C07294=1020.176,319.167,359.790,170.598,49.800,159.708
C07295=1020.170,318.918,359.824,170.593,49.803,159.708
C07296=1020.163,318.671,359.858,170.586,49.806,159.708
C07297=1020.156,318.424,359.891,170.580,49.809,159.707
C07298=1020.149,318.176,359.925,170.574,49.812,159.707
C07299=1020.143,317.928,359.959,170.568,49.814,159.707
C07300=1020.136,317.681,359.993,170.563,49.818,159.706
C07301=1020.129,317.433,360.027,170.556,49.821,159.706
C07302=1020.122,317.186,360.060,170.551,49.823,159.706
C07303=1020.116,316.938,360.094,170.545,49.826,159.705
C07304=1020.109,316.690,360.128,170.538,49.829,159.705
C07305=1020.102,316.443,360.161,170.533,49.832,159.705
C07306=1020.095,316.195,360.195,170.527,49.835,159.705
C07307=1020.089,315.947,360.229,170.521,49.838,159.704
C07308=1020.083,315.700,360.262,170.515,49.840,159.704
C07309=1020.075,315.452,360.296,170.510,49.844,159.704
C07310=1020.069,315.205,360.329,170.503,49.847,159.704
C07311=1020.063,314.957,360.363,170.497,49.849,159.703
C07312=1020.056,314.710,360.396,170.492,49.853,159.703
C07313=1020.049,314.462,360.430,170.485,49.855,159.703
C07314=1020.042,314.214,360.463,170.480,49.858,159.702
C07315=1020.036,313.966,360.497,170.474,49.861,159.702
C07316=1020.030,313.719,360.530,170.468,49.864,159.702
C07317=1020.023,313.471,360.564,170.462,49.867,159.702
C07318=1020.016,313.224,360.597,170.457,49.870,159.702
C07319=1020.010,312.975,360.631,170.451,49.873,159.701
C07320=1020.003,312.729,360.665,170.445,49.877,159.701
C07321=1019.997,312.481,360.697,170.439,49.879,159.701
C07322=1019.990,312.233,360.731,170.434,49.883,159.701
C07323=1019.983,311.986,360.764,170.427,49.886,159.700
C07324=1019.978,311.738,360.798,170.422,49.889,159.700
C07325=1019.971,311.490,360.831,170.416,49.891,159.700
C07326=1019.964,311.243,360.865,170.411,49.895,159.700
C07327=1019.957,310.995,360.898,170.404,49.898,159.699
C07328=1019.952,310.747,360.931,170.399,49.901,159.699
C07329=1019.945,310.500,360.964,170.393,49.904,159.699
C07330=1019.938,310.252,360.998,170.388,49.907,159.699
C07331=1019.932,310.004,361.030,170.382,49.910,159.699
C07332=1019.925,309.757,361.064,170.376,49.913,159.698
C07333=1019.918,309.509,361.097,170.371,49.917,159.698
C07334=1019.911,309.262,361.129,170.365,49.920,159.698
C07335=1019.905,309.014,361.162,170.359,49.923,159.698
C07336=1019.897,308.766,361.194,170.353,49.927,159.698
C07337=1019.891,308.523,361.226,170.347,49.930,159.698
C07338=1019.885,308.281,361.258,170.342,49.933,159.697
C07339=1019.878,308.039,361.290,170.337,49.936,159.697
C07340=1019.871,307.796,361.322,170.332,49.940,159.697
C07341=1019.864,307.553,361.353,170.325,49.943,159.697
C07342=1019.858,307.311,361.385,170.320,49.947,159.697
C07343=1019.852,307.069,361.418,170.315,49.950,159.697
C07344=1019.845,306.827,361.449,170.309,49.953,159.697
C07345=1019.839,306.579,361.481,170.303,49.957,159.697
C07346=1019.831,306.331,361.514,170.298,49.960,159.696
C07347=1019.825,306.083,361.547,170.293,49.963,159.696
C07348=1019.819,305.836,361.579,170.286,49.967,159.696
C07349=1019.812,305.588,361.611,170.281,49.970,159.696
C07350=1019.806,305.340,361.643,170.276,49.974,159.696
C07351=1019.798,305.092,361.676,170.269,49.977,159.696
C07352=1019.792,304.845,361.709,170.264,49.981,159.696
C07353=1019.785,304.597,361.741,170.259,49.984,159.696
C07354=1019.779,304.349,361.773,170.253,49.987,159.695
C07355=1019.772,304.102,361.806,170.247,49.991,159.695
C07356=1019.765,303.854,361.838,170.242,49.995,159.695
C07357=1019.759,303.605,361.870,170.236,49.998,159.695
C07358=1019.752,303.358,361.903,170.231,50.002,159.695
C07359=1019.745,303.110,361.935,170.226,50.005,159.695
C07360=1019.739,302.862,361.967,170.219,50.009,159.695
C07361=1019.732,302.615,361.999,170.214,50.013,159.695
C07362=1019.726,302.367,362.031,170.209,50.016,159.695
C07363=1019.719,302.119,362.063,170.204,50.019,159.695
C07364=1019.713,301.872,362.096,170.198,50.023,159.694
C07365=1019.707,301.624,362.128,170.192,50.026,159.694
C07366=1019.699,301.376,362.161,170.187,50.030,159.694
C07367=1019.693,301.127,362.193,170.181,50.034,159.694
C07368=1019.686,300.880,362.225,170.176,50.037,159.694
C07369=1019.680,300.632,362.257,170.171,50.041,159.694
C07370=1019.674,300.384,362.288,170.165,50.045,159.694
C07371=1019.667,300.136,362.321,170.159,50.048,159.694
C07372=1019.661,299.888,362.353,170.154,50.052,159.694
C07373=1019.654,299.641,362.385,170.149,50.055,159.694
C07374=1019.648,299.393,362.417,170.143,50.059,159.694
C07375=1019.641,299.145,362.449,170.138,50.063,159.694
C07376=1019.635,298.897,362.481,170.133,50.066,159.694
C07377=1019.629,298.650,362.513,170.128,50.070,159.694
C07378=1019.623,298.402,362.545,170.121,50.074,159.694
C07379=1019.617,298.154,362.577,170.116,50.077,159.693
C07380=1019.610,297.906,362.609,170.111,50.081,159.694
C07381=1019.604,297.658,362.641,170.106,50.084,159.693
C07382=1019.597,297.411,362.673,170.100,50.089,159.693
C07383=1019.591,297.163,362.705,170.095,50.092,159.693
C07384=1019.585,296.915,362.736,170.090,50.096,159.693
C07385=1019.579,296.667,362.768,170.084,50.100,159.693
C07386=1019.572,296.419,362.801,170.079,50.104,159.693
C07387=1019.566,296.172,362.832,170.073,50.107,159.693
C07388=1019.560,295.924,362.864,170.069,50.111,159.693
C07389=1019.553,295.676,362.896,170.063,50.115,159.693
C07390=1019.547,295.427,362.928,170.057,50.118,159.693
C07391=1019.541,295.179,362.959,170.052,50.122,159.693
C07392=1019.535,294.933,362.991,170.047,50.126,159.693
C07393=1019.529,294.684,363.024,170.042,50.130,159.693
C07394=1019.522,294.436,363.055,170.036,50.134,159.693
C07395=1019.516,294.188,363.087,170.031,50.137,159.693
C07396=1019.510,293.940,363.118,170.026,50.141,159.693
C07397=1019.504,293.707,363.147,170.021,50.145,159.693
C07398=1019.499,293.473,363.178,170.016,50.149,159.693
C07399=1019.492,293.240,363.208,170.011,50.152,159.693
C07400=1019.486,293.006,363.238,170.006,50.156,159.693
C07401=1019.481,292.772,363.267,170.001,50.160,159.693
C07402=1019.475,292.539,363.297,169.996,50.163,159.693
C07403=1019.469,292.305,363.326,169.992,50.167,159.693
C07404=1019.462,292.072,363.356,169.987,50.171,159.693
C07405=1019.457,291.823,363.387,169.981,50.175,159.693
C07406=1019.450,291.575,363.418,169.976,50.179,159.694
C07407=1019.443,291.328,363.450,169.971,50.183,159.694
C07408=1019.437,291.080,363.481,169.965,50.187,159.694
C07409=1019.431,290.832,363.512,169.960,50.191,159.694
C07410=1019.424,290.584,363.543,169.955,50.195,159.694
C07411=1019.419,290.336,363.574,169.951,50.199,159.694
C07412=1019.412,290.088,363.605,169.945,50.204,159.694
C07413=1019.405,289.840,363.637,169.940,50.208,159.694
C07414=1019.400,289.592,363.667,169.935,50.212,159.694
C07415=1019.393,289.344,363.699,169.929,50.216,159.694
C07416=1019.386,289.096,363.729,169.924,50.220,159.694
C07417=1019.380,288.849,363.760,169.919,50.224,159.694
C07418=1019.374,288.601,363.792,169.913,50.228,159.694
C07419=1019.367,288.352,363.823,169.908,50.232,159.694
C07420=1019.361,288.105,363.854,169.903,50.236,159.694
C07421=1019.355,287.856,363.884,169.899,50.240,159.694
C07422=1019.348,287.608,363.916,169.893,50.245,159.694
C07423=1019.342,287.361,363.946,169.888,50.249,159.695
C07424=1019.336,287.112,363.977,169.883,50.253,159.695
C07425=1019.329,286.865,364.008,169.877,50.258,159.695
C07426=1019.323,286.616,364.039,169.872,50.262,159.695
C07427=1019.316,286.369,364.070,169.868,50.265,159.695
C07428=1019.311,286.121,364.100,169.863,50.270,159.695
C07429=1019.304,285.872,364.131,169.857,50.274,159.695
C07430=1019.298,285.625,364.162,169.852,50.278,159.695
C07431=1019.292,285.376,364.193,169.847,50.282,159.695
C07432=1019.286,285.129,364.223,169.842,50.287,159.696
C07433=1019.279,284.881,364.255,169.837,50.291,159.696
C07434=1019.273,284.633,364.285,169.832,50.295,159.696
C07435=1019.267,284.384,364.316,169.827,50.300,159.696
C07436=1019.261,284.137,364.346,169.822,50.304,159.696
C07437=1019.255,283.888,364.377,169.817,50.309,159.696
C07438=1019.248,283.641,364.407,169.811,50.313,159.696
C07439=1019.242,283.392,364.437,169.807,50.318,159.697
C07440=1019.235,283.145,364.468,169.802,50.322,159.697
C07441=1019.229,282.896,364.499,169.796,50.327,159.697
C07442=1019.222,282.649,364.529,169.791,50.331,159.697
C07443=1019.216,282.400,364.560,169.787,50.336,159.697
C07444=1019.210,282.152,364.590,169.782,50.340,159.697
C07445=1019.204,281.904,364.621,169.776,50.345,159.698
C07446=1019.197,281.656,364.650,169.772,50.349,159.698
C07447=1019.191,281.409,364.681,169.767,50.353,159.698
C07448=1019.185,281.160,364.711,169.761,50.358,159.698
C07449=1019.179,280.912,364.742,169.757,50.362,159.698
C07450=1019.173,280.664,364.772,169.752,50.366,159.698
C07451=1019.166,280.416,364.802,169.746,50.371,159.698
C07452=1019.160,280.168,364.833,169.742,50.376,159.699
C07453=1019.154,279.920,364.863,169.737,50.380,159.699
C07454=1019.148,279.671,364.893,169.731,50.385,159.699
C07455=1019.141,279.423,364.923,169.726,50.389,159.699
C07456=1019.136,279.175,364.953,169.722,50.394,159.699
C07457=1019.130,278.948,364.981,169.717,50.398,159.699
C07458=1019.124,278.721,365.009,169.713,50.402,159.700
C07459=1019.119,278.493,365.037,169.708,50.406,159.700
C07460=1019.113,278.265,365.064,169.704,50.411,159.700
C07461=1019.108,278.038,365.092,169.699,50.415,159.700
C07462=1019.102,277.810,365.120,169.694,50.419,159.700
C07463=1019.096,277.583,365.148,169.690,50.423,159.701
C07464=1019.090,277.355,365.175,169.685,50.427,159.701
C07465=1019.084,277.107,365.205,169.681,50.432,159.701
C07466=1019.079,276.859,365.235,169.676,50.437,159.701
C07467=1019.073,276.611,365.266,169.672,50.441,159.702
C07468=1019.066,276.363,365.295,169.666,50.446,159.702
C07469=1019.060,276.115,365.326,169.661,50.450,159.702
C07470=1019.054,275.867,365.355,169.657,50.455,159.702
C07471=1019.047,275.618,365.385,169.651,50.460,159.702
C07472=1019.041,275.371,365.415,169.647,50.465,159.703
C07473=1019.035,275.122,365.445,169.641,50.470,159.703
C07474=1019.029,274.875,365.475,169.637,50.475,159.703
C07475=1019.023,274.626,365.505,169.632,50.479,159.703
C07476=1019.016,274.378,365.534,169.627,50.484,159.704
C07477=1019.011,274.130,365.564,169.622,50.489,159.704
C07478=1019.004,273.882,365.594,169.618,50.494,159.704
C07479=1018.999,273.634,365.623,169.612,50.499,159.704
C07480=1018.991,273.385,365.653,169.608,50.503,159.705
C07481=1018.986,273.137,365.683,169.603,50.508,159.705
C07482=1018.979,272.889,365.713,169.598,50.513,159.705
C07483=1018.974,272.641,365.742,169.593,50.518,159.705
C07484=1018.968,272.393,365.771,169.589,50.522,159.706
C07485=1018.962,272.145,365.802,169.583,50.527,159.706
C07486=1018.955,271.896,365.831,169.579,50.532,159.706
C07487=1018.949,271.648,365.860,169.575,50.537,159.707
C07488=1018.943,271.400,365.891,169.569,50.542,159.707
C07489=1018.937,271.152,365.920,169.565,50.547,159.707
C07490=1018.931,270.904,365.949,169.560,50.552,159.707
C07491=1018.925,270.656,365.979,169.555,50.557,159.707
C07492=1018.918,270.408,366.008,169.550,50.562,159.708
C07493=1018.913,270.160,366.038,169.545,50.567,159.708
C07494=1018.906,269.911,366.067,169.540,50.572,159.708
C07495=1018.900,269.662,366.097,169.536,50.577,159.709
C07496=1018.894,269.415,366.127,169.530,50.582,159.709
C07497=1018.888,269.167,366.156,169.526,50.587,159.709
C07498=1018.882,268.918,366.185,169.522,50.592,159.710
C07499=1018.876,268.670,366.214,169.516,50.597,159.710
C07500=1018.870,268.422,366.243,169.512,50.602,159.710
C07501=1018.863,268.174,366.272,169.507,50.607,159.710
C07502=1018.858,267.925,366.302,169.502,50.612,159.711
C07503=1018.852,267.677,366.331,169.498,50.617,159.711
C07504=1018.845,267.429,366.360,169.493,50.622,159.711
C07505=1018.839,267.181,366.389,169.488,50.627,159.712
C07506=1018.834,266.933,366.419,169.484,50.632,159.712
C07507=1018.827,266.684,366.448,169.479,50.637,159.712
C07508=1018.821,266.436,366.477,169.474,50.643,159.713
C07509=1018.815,266.188,366.506,169.469,50.648,159.713
C07510=1018.809,265.940,366.535,169.465,50.653,159.714
C07511=1018.803,265.692,366.565,169.460,50.658,159.714
C07512=1018.797,265.443,366.594,169.455,50.664,159.714
C07513=1018.791,265.195,366.623,169.451,50.668,159.714
C07514=1018.784,264.947,366.652,169.446,50.674,159.715
C07515=1018.778,264.699,366.681,169.441,50.679,159.715
C07516=1018.772,264.451,366.710,169.437,50.684,159.716
C07517=1018.767,264.226,366.736,169.433,50.689,159.716
C07518=1018.762,264.000,366.762,169.428,50.693,159.716
C07519=1018.755,263.775,366.788,169.424,50.698,159.716
C07520=1018.750,263.550,366.815,169.419,50.703,159.717
C07521=1018.745,263.324,366.841,169.415,50.708,159.717
C07522=1018.739,263.099,366.866,169.412,50.713,159.718
C07523=1018.734,262.875,366.893,169.407,50.717,159.718
C07524=1018.728,262.649,366.919,169.403,50.722,159.718
C07525=1018.722,262.400,366.948,169.398,50.728,159.718
C07526=1018.717,262.153,366.977,169.393,50.733,159.719
C07527=1018.710,261.904,367.006,169.389,50.738,159.719
C07528=1018.704,261.656,367.034,169.384,50.744,159.720
C07529=1018.698,261.408,367.063,169.380,50.749,159.720
C07530=1018.692,261.159,367.093,169.375,50.755,159.720
C07531=1018.686,260.911,367.121,169.370,50.759,159.721
C07532=1018.680,260.662,367.150,169.366,50.765,159.721
C07533=1018.674,260.415,367.179,169.361,50.771,159.722
C07534=1018.668,260.166,367.207,169.357,50.776,159.722
C07535=1018.662,259.918,367.236,169.352,50.781,159.722
C07536=1018.656,259.669,367.264,169.347,50.786,159.723
C07537=1018.649,259.422,367.293,169.342,50.792,159.723
C07538=1018.643,259.173,367.321,169.338,50.798,159.724
C07539=1018.638,258.925,367.349,169.333,50.803,159.724
C07540=1018.631,258.677,367.377,169.329,50.809,159.724
C07541=1018.625,258.428,367.406,169.324,50.814,159.725
C07542=1018.619,258.179,367.434,169.320,50.820,159.725
C07543=1018.612,257.932,367.463,169.315,50.826,159.726
C07544=1018.606,257.683,367.491,169.311,50.832,159.726
C07545=1018.601,257.435,367.519,169.306,50.837,159.727
C07546=1018.594,257.187,367.547,169.301,50.843,159.727
C07547=1018.588,256.938,367.576,169.297,50.848,159.728
C07548=1018.582,256.690,367.604,169.292,50.854,159.728
C07549=1018.575,256.441,367.632,169.288,50.860,159.729
C07550=1018.570,256.193,367.660,169.283,50.865,159.729
C07551=1018.563,255.945,367.689,169.279,50.871,159.729
C07552=1018.557,255.696,367.716,169.273,50.877,159.730
C07553=1018.551,255.448,367.745,169.269,50.882,159.730
C07554=1018.545,255.200,367.773,169.265,50.888,159.731
C07555=1018.539,254.951,367.800,169.261,50.894,159.731
C07556=1018.533,254.703,367.829,169.256,50.900,159.732
C07557=1018.527,254.455,367.857,169.252,50.905,159.732
C07558=1018.521,254.207,367.885,169.246,50.911,159.733
C07559=1018.515,253.958,367.913,169.243,50.917,159.733
C07560=1018.508,253.709,367.941,169.238,50.923,159.734
C07561=1018.503,253.461,367.969,169.234,50.928,159.734
C07562=1018.497,253.213,367.997,169.229,50.934,159.734
C07563=1018.490,252.964,368.025,169.224,50.940,159.735
C07564=1018.485,252.716,368.053,169.220,50.946,159.736
C07565=1018.479,252.467,368.081,169.215,50.951,159.736
C07566=1018.472,252.220,368.110,169.211,50.957,159.736
C07567=1018.466,251.972,368.138,169.206,50.963,159.737
C07568=1018.460,251.723,368.166,169.202,50.969,159.737
C07569=1018.454,251.475,368.194,169.197,50.974,159.738
C07570=1018.448,251.226,368.222,169.193,50.980,159.738
C07571=1018.442,250.977,368.250,169.188,50.986,159.739
C07572=1018.436,250.730,368.278,169.184,50.992,159.739
C07573=1018.431,250.480,368.305,169.179,50.998,159.740
C07574=1018.425,250.233,368.333,169.175,51.003,159.740
C07575=1018.419,249.984,368.361,169.171,51.010,159.741
C07576=1018.413,249.735,368.389,169.167,51.015,159.741
C07577=1018.407,249.510,368.414,169.163,51.021,159.742
C07578=1018.402,249.284,368.440,169.158,51.026,159.742
C07579=1018.396,249.057,368.465,169.154,51.032,159.743
C07580=1018.392,248.831,368.491,169.150,51.037,159.743
C07581=1018.386,248.605,368.516,169.146,51.042,159.744
C07582=1018.381,248.379,368.541,169.142,51.048,159.744
C07583=1018.375,248.154,368.566,169.138,51.053,159.745
C07584=1018.370,247.927,368.592,169.134,51.059,159.745
C07585=1018.364,247.679,368.620,169.129,51.065,159.746
C07586=1018.358,247.430,368.647,169.125,51.071,159.746
C07587=1018.353,247.182,368.675,169.120,51.076,159.747
C07588=1018.346,246.934,368.703,169.117,51.083,159.747
C07589=1018.341,246.685,368.731,169.112,51.088,159.748
C07590=1018.334,246.437,368.759,169.108,51.094,159.748
C07591=1018.329,246.188,368.786,169.103,51.100,159.749
C07592=1018.323,245.940,368.814,169.098,51.107,159.749
C07593=1018.317,245.692,368.842,169.094,51.112,159.750
C07594=1018.311,245.443,368.869,169.090,51.119,159.750
C07595=1018.306,245.194,368.897,169.085,51.124,159.751
C07596=1018.300,244.947,368.925,169.081,51.130,159.751
C07597=1018.294,244.698,368.953,169.077,51.137,159.752
C07598=1018.288,244.450,368.979,169.072,51.142,159.753
C07599=1018.282,244.201,369.008,169.068,51.148,159.753
C07600=1018.277,243.953,369.036,169.064,51.155,159.754
C07601=1018.271,243.704,369.062,169.060,51.160,159.754
C07602=1018.265,243.456,369.091,169.055,51.167,159.755
C07603=1018.259,243.208,369.118,169.050,51.173,159.755
C07604=1018.254,242.959,369.146,169.046,51.179,159.756
C07605=1018.247,242.711,369.173,169.042,51.185,159.756
C07606=1018.242,242.462,369.200,169.038,51.191,159.757
C07607=1018.236,242.214,369.228,169.034,51.198,159.758
C07608=1018.230,241.965,369.255,169.029,51.204,159.758
C07609=1018.222,241.657,369.289,169.024,51.212,159.759
C07610=1018.216,241.348,369.323,169.018,51.219,159.760
C07611=1018.208,241.040,369.357,169.014,51.227,159.761
C07612=1018.201,240.731,369.390,169.007,51.235,159.761
C07613=1018.195,240.483,369.418,169.004,51.241,159.762
C07614=1018.189,240.233,369.445,168.999,51.248,159.762
C07615=1018.183,239.985,369.472,168.994,51.254,159.763
C07616=1018.177,239.737,369.499,168.991,51.261,159.764
C07617=1018.172,239.489,369.526,168.986,51.267,159.764
C07618=1018.166,239.240,369.553,168.981,51.274,159.765
C07619=1018.160,238.992,369.581,168.978,51.280,159.766
C07620=1018.154,238.743,369.607,168.973,51.286,159.766
C07621=1018.148,238.494,369.634,168.969,51.293,159.767
C07622=1018.143,238.246,369.662,168.965,51.299,159.767
C07623=1018.137,237.998,369.689,168.960,51.305,159.768
C07624=1018.130,237.749,369.716,168.956,51.312,159.769
C07625=1018.124,237.501,369.743,168.951,51.318,159.769
C07626=1018.119,237.252,369.769,168.947,51.324,159.770
C07627=1018.113,237.004,369.796,168.943,51.332,159.771
C07628=1018.107,236.755,369.823,168.939,51.338,159.771
C07629=1018.101,236.506,369.850,168.934,51.345,159.772
C07630=1018.095,236.258,369.876,168.930,51.351,159.772
C07631=1018.089,236.010,369.903,168.926,51.357,159.773
C07632=1018.083,235.761,369.931,168.921,51.364,159.774
C07633=1018.077,235.513,369.957,168.918,51.371,159.775
C07634=1018.071,235.265,369.984,168.913,51.377,159.775
C07635=1018.065,235.016,370.011,168.909,51.384,159.776
C07636=1018.059,234.767,370.038,168.904,51.391,159.776
C07637=1018.049,234.368,370.080,168.897,51.401,159.777
C07638=1018.040,233.970,370.124,168.891,51.412,159.779
C07639=1018.031,233.571,370.166,168.884,51.422,159.780
C07640=1018.022,233.173,370.208,168.877,51.433,159.781
C07641=1018.015,232.924,370.235,168.873,51.440,159.781
C07642=1018.010,232.676,370.261,168.868,51.447,159.782
C07643=1018.004,232.428,370.288,168.865,51.453,159.783
C07644=1017.998,232.179,370.315,168.861,51.460,159.784
C07645=1017.992,231.931,370.341,168.856,51.466,159.784
C07646=1017.986,231.682,370.368,168.852,51.474,159.785
C07647=1017.981,231.434,370.395,168.847,51.480,159.785
C07648=1017.975,231.184,370.421,168.844,51.487,159.786
C07649=1017.969,230.936,370.448,168.839,51.494,159.787
C07650=1017.963,230.688,370.474,168.835,51.500,159.788
C07651=1017.957,230.439,370.501,168.831,51.507,159.788
C07652=1017.952,230.191,370.528,168.826,51.514,159.789
C07653=1017.946,229.942,370.553,168.823,51.521,159.790
C07654=1017.940,229.694,370.580,168.818,51.527,159.790
C07655=1017.935,229.445,370.607,168.814,51.534,159.791
C07656=1017.929,229.197,370.633,168.810,51.542,159.792
C07657=1017.923,228.948,370.659,168.805,51.548,159.792
C07658=1017.917,228.700,370.685,168.802,51.555,159.793
C07659=1017.911,228.452,370.712,168.797,51.562,159.794
C07660=1017.906,228.203,370.738,168.793,51.569,159.795
C07661=1017.899,227.953,370.765,168.789,51.576,159.796
C07662=1017.893,227.705,370.792,168.784,51.582,159.796
C07663=1017.887,227.456,370.817,168.780,51.590,159.797
C07664=1017.881,227.208,370.844,168.776,51.597,159.798
C07665=1017.876,226.959,370.870,168.772,51.603,159.798
C07666=1017.870,226.711,370.896,168.768,51.610,159.799
C07667=1017.864,226.462,370.923,168.764,51.618,159.800
C07668=1017.858,226.214,370.948,168.760,51.625,159.801
C07669=1017.852,225.965,370.975,168.756,51.632,159.802
C07670=1017.846,225.717,371.000,168.751,51.639,159.802
C07671=1017.841,225.468,371.026,168.747,51.646,159.803
C07672=1017.835,225.219,371.053,168.743,51.653,159.804
C07673=1017.829,224.971,371.078,168.739,51.660,159.804
C07674=1017.823,224.722,371.105,168.734,51.667,159.805
C07675=1017.817,224.474,371.130,168.730,51.675,159.806
C07676=1017.811,224.225,371.156,168.726,51.682,159.807
C07677=1017.806,223.976,371.183,168.723,51.689,159.808
C07678=1017.799,223.728,371.208,168.719,51.696,159.809
C07679=1017.794,223.479,371.234,168.714,51.703,159.809
C07680=1017.788,223.231,371.260,168.710,51.710,159.810
C07681=1017.782,222.982,371.286,168.706,51.717,159.811
C07682=1017.776,222.734,371.311,168.702,51.724,159.811
C07683=1017.771,222.485,371.338,168.698,51.732,159.812
C07684=1017.765,222.236,371.363,168.693,51.739,159.813
C07685=1017.759,221.988,371.389,168.689,51.746,159.814
C07686=1017.753,221.739,371.415,168.685,51.753,159.815
C07687=1017.747,221.491,371.441,168.681,51.761,159.815
C07688=1017.741,221.242,371.467,168.677,51.768,159.816
C07689=1017.735,220.993,371.492,168.673,51.775,159.817
C07690=1017.729,220.745,371.519,168.669,51.783,159.818
C07691=1017.725,220.496,371.544,168.665,51.790,159.819
C07692=1017.718,220.248,371.570,168.661,51.798,159.820
C07693=1017.712,220.014,371.594,168.657,51.804,159.820
C07694=1017.707,219.781,371.618,168.653,51.811,159.821
C07695=1017.702,219.548,371.642,168.649,51.818,159.822
C07696=1017.697,219.313,371.667,168.645,51.824,159.822
C07697=1017.691,219.080,371.691,168.641,51.832,159.823
C07698=1017.686,218.847,371.715,168.638,51.839,159.824
C07699=1017.681,218.613,371.739,168.633,51.845,159.825
C07700=1017.675,218.379,371.764,168.630,51.852,159.826
C07701=1017.669,218.131,371.790,168.626,51.859,159.826
C07702=1017.664,217.883,371.815,168.622,51.867,159.827
C07703=1017.657,217.634,371.840,168.617,51.875,159.828
C07704=1017.651,217.385,371.865,168.613,51.882,159.829
C07705=1017.646,217.136,371.891,168.609,51.890,159.830
C07706=1017.640,216.888,371.916,168.605,51.897,159.831
C07707=1017.634,216.640,371.942,168.601,51.905,159.831
C07708=1017.628,216.391,371.967,168.597,51.913,159.832
C07709=1017.622,216.142,371.993,168.593,51.920,159.833
C07710=1017.616,215.893,372.018,168.589,51.927,159.834
C07711=1017.610,215.645,372.043,168.585,51.935,159.835
C07712=1017.605,215.396,372.068,168.581,51.942,159.836
C07713=1017.599,215.147,372.094,168.576,51.951,159.837
C07714=1017.593,214.898,372.119,168.572,51.958,159.838
C07715=1017.587,214.650,372.144,168.569,51.966,159.839
C07716=1017.582,214.401,372.170,168.565,51.973,159.839
C07717=1017.576,214.153,372.195,168.561,51.981,159.840
C07718=1017.569,213.904,372.221,168.557,51.989,159.841
C07719=1017.564,213.656,372.246,168.553,51.996,159.842
C07720=1017.559,213.407,372.271,168.549,52.004,159.843
C07721=1017.552,213.158,372.296,168.544,52.012,159.844
C07722=1017.546,212.909,372.321,168.540,52.019,159.845
C07723=1017.541,212.661,372.347,168.536,52.027,159.846
C07724=1017.535,212.412,372.372,168.532,52.035,159.846
C07725=1017.529,212.163,372.397,168.529,52.043,159.847
C07726=1017.524,211.915,372.422,168.524,52.050,159.848
C07727=1017.518,211.666,372.448,168.521,52.058,159.849
C07728=1017.512,211.417,372.473,168.516,52.066,159.850
C07729=1017.507,211.169,372.497,168.512,52.074,159.851
C07730=1017.500,210.920,372.523,168.508,52.082,159.852
C07731=1017.495,210.671,372.549,168.504,52.089,159.853
C07732=1017.489,210.423,372.574,168.500,52.097,159.854
C07733=1017.483,210.174,372.598,168.496,52.104,159.854
C07734=1017.477,209.925,372.624,168.493,52.112,159.855
C07735=1017.472,209.677,372.649,168.488,52.121,159.856
C07736=1017.466,209.428,372.674,168.484,52.128,159.857
C07737=1017.461,209.180,372.699,168.480,52.136,159.858
C07738=1017.455,208.930,372.723,168.477,52.144,159.859
C07739=1017.449,208.682,372.749,168.472,52.152,159.860
C07740=1017.443,208.434,372.774,168.468,52.160,159.861
C07741=1017.437,208.184,372.798,168.464,52.168,159.862
C07742=1017.431,207.936,372.824,168.460,52.176,159.863
C07743=1017.426,207.687,372.848,168.456,52.184,159.864
C07744=1017.420,207.438,372.873,168.452,52.192,159.865
C07745=1017.414,207.190,372.898,168.448,52.200,159.866
C07746=1017.408,206.941,372.923,168.445,52.208,159.867
C07747=1017.403,206.693,372.947,168.440,52.216,159.868
C07748=1017.397,206.444,372.972,168.436,52.224,159.868
C07749=1017.391,206.195,372.997,168.432,52.232,159.869
C07750=1017.385,205.947,373.022,168.429,52.240,159.870
C07751=1017.379,205.697,373.047,168.424,52.248,159.871
C07752=1017.374,205.449,373.071,168.420,52.256,159.872
C07753=1017.369,205.212,373.095,168.417,52.264,159.873
C07754=1017.362,204.975,373.118,168.413,52.271,159.874
C07755=1017.357,204.739,373.141,168.409,52.280,159.875
C07756=1017.352,204.503,373.164,168.405,52.288,159.876
C07757=1017.346,204.265,373.188,168.401,52.295,159.877
C07758=1017.340,204.029,373.211,168.398,52.303,159.878
C07759=1017.335,203.793,373.235,168.394,52.311,159.879
C07760=1017.330,203.556,373.258,168.390,52.319,159.880
C07761=1017.305,202.315,373.374,167.903,52.236,159.767
C07762=1017.300,202.066,373.396,167.898,52.246,159.768
C07763=1017.296,201.818,373.419,167.894,52.255,159.769
C07764=1017.291,201.570,373.442,167.889,52.264,159.770
C07765=1017.286,201.321,373.465,167.884,52.273,159.771
C07766=1017.281,201.072,373.487,167.880,52.282,159.772
C07767=1017.276,200.823,373.511,167.875,52.291,159.773
C07768=1017.272,200.573,373.533,167.870,52.301,159.774
C07769=1017.267,200.325,373.556,167.866,52.310,159.775
C07770=1017.262,200.077,373.579,167.861,52.319,159.776
C07771=1017.257,199.827,373.602,167.857,52.329,159.778
C07772=1017.253,199.578,373.625,167.852,52.338,159.779
C07773=1017.248,199.329,373.647,167.848,52.348,159.780
C07774=1017.243,199.080,373.671,167.843,52.357,159.781
C07775=1017.238,198.831,373.693,167.838,52.366,159.782
C07776=1017.233,198.583,373.715,167.834,52.376,159.783
C07777=1017.229,198.333,373.738,167.829,52.385,159.784
C07778=1017.223,198.085,373.761,167.825,52.395,159.785
C07779=1017.218,197.836,373.783,167.820,52.405,159.786
C07780=1017.214,197.587,373.805,167.816,52.414,159.787
C07781=1017.208,197.338,373.828,167.811,52.423,159.788
C07782=1017.203,197.089,373.850,167.806,52.433,159.789
C07783=1017.199,196.840,373.872,167.802,52.442,159.790
C07784=1017.194,196.591,373.895,167.797,52.452,159.791
C07785=1017.189,196.342,373.917,167.793,52.461,159.792
C07786=1017.184,196.093,373.939,167.789,52.471,159.794
C07787=1017.179,195.844,373.963,167.784,52.480,159.795
C07788=1017.174,195.595,373.985,167.780,52.490,159.796
C07789=1017.169,195.346,374.006,167.776,52.499,159.797
C07790=1017.165,195.097,374.029,167.770,52.509,159.798
C07791=1017.159,194.848,374.052,167.766,52.518,159.799
C07792=1017.155,194.600,374.074,167.762,52.528,159.800
C07793=1017.151,194.350,374.096,167.757,52.537,159.801
C07794=1017.145,194.101,374.118,167.753,52.547,159.802
C07795=1017.140,193.853,374.141,167.749,52.557,159.803
C07796=1017.135,193.604,374.163,167.744,52.566,159.804
C07797=1017.131,193.355,374.185,167.739,52.575,159.805
C07798=1017.126,193.105,374.207,167.736,52.585,159.807
C07799=1017.121,192.856,374.229,167.730,52.595,159.807
C07800=1017.117,192.607,374.252,167.726,52.604,159.809
C07801=1017.112,192.359,374.274,167.722,52.613,159.810
C07802=1017.106,192.110,374.297,167.718,52.623,159.811
C07803=1017.101,191.861,374.318,167.713,52.632,159.812
C07804=1017.097,191.612,374.341,167.709,52.642,159.813
C07805=1017.092,191.363,374.363,167.705,52.651,159.814
C07806=1017.088,191.114,374.385,167.701,52.661,159.815
C07807=1017.083,190.864,374.407,167.695,52.670,159.816
C07808=1017.078,190.615,374.429,167.692,52.680,159.817
C07809=1017.073,190.367,374.452,167.687,52.689,159.818
C07810=1017.069,190.118,374.474,167.683,52.698,159.819
C07811=1017.064,189.869,374.496,167.678,52.709,159.821
C07812=1017.059,189.620,374.518,167.674,52.718,159.822
C07813=1017.054,189.372,374.540,167.670,52.727,159.823
C07814=1017.050,189.122,374.563,167.666,52.737,159.824
C07815=1017.045,188.873,374.585,167.661,52.747,159.825
C07816=1017.040,188.624,374.607,167.657,52.756,159.826
C07817=1017.035,188.375,374.628,167.653,52.766,159.827
C07818=1017.031,188.126,374.651,167.649,52.775,159.828
C07819=1017.026,187.877,374.673,167.645,52.784,159.829
C07820=1017.022,187.629,374.695,167.640,52.794,159.830
C07821=1017.017,187.348,374.720,167.635,52.805,159.832
C07822=1017.011,187.068,374.745,167.631,52.816,159.833
C07823=1017.007,186.787,374.769,167.626,52.826,159.834
C07824=1017.001,186.507,374.794,167.622,52.837,159.836
C07825=1016.996,186.258,374.815,167.616,52.847,159.836
C07826=1016.992,186.009,374.837,167.612,52.856,159.838
C07827=1016.987,185.760,374.860,167.608,52.866,159.839
C07828=1016.983,185.511,374.881,167.604,52.875,159.840
C07829=1016.978,185.262,374.903,167.600,52.884,159.841
C07830=1016.974,185.013,374.926,167.596,52.894,159.842
C07831=1016.969,184.764,374.948,167.592,52.903,159.843
C07832=1016.964,184.516,374.970,167.588,52.913,159.844
C07833=1016.959,184.267,374.991,167.583,52.923,159.845
C07834=1016.955,184.017,375.013,167.579,52.932,159.846
C07835=1016.951,183.768,375.035,167.575,52.941,159.847
C07836=1016.946,183.519,375.057,167.571,52.951,159.849
C07837=1016.941,183.270,375.079,167.567,52.961,159.850
C07838=1016.937,183.021,375.101,167.563,52.970,159.851
C07839=1016.932,182.772,375.122,167.559,52.980,159.852
C07840=1016.928,182.523,375.144,167.555,52.989,159.853
C07841=1016.924,182.274,375.167,167.551,52.998,159.854
C07842=1016.919,182.025,375.189,167.547,53.008,159.856
C07843=1016.914,181.776,375.210,167.543,53.017,159.857
C07844=1016.909,181.527,375.232,167.538,53.028,159.858
C07845=1016.904,181.278,375.252,167.534,53.037,159.859
C07846=1016.899,181.029,375.274,167.530,53.047,159.860
C07847=1016.895,180.780,375.295,167.526,53.057,159.861
C07848=1016.889,180.530,375.316,167.522,53.067,159.862
C07849=1016.885,180.282,375.338,167.518,53.077,159.864
C07850=1016.880,180.032,375.359,167.514,53.086,159.865
C07851=1016.875,179.784,375.380,167.509,53.096,159.866
C07852=1016.870,179.534,375.401,167.505,53.106,159.867
C07853=1016.865,179.285,375.422,167.501,53.115,159.868
C07854=1016.860,179.036,375.444,167.498,53.125,159.869
C07855=1016.855,178.787,375.465,167.493,53.136,159.871
C07856=1016.850,178.538,375.485,167.489,53.145,159.872
C07857=1016.845,178.289,375.507,167.485,53.155,159.873
C07858=1016.841,178.039,375.528,167.481,53.165,159.874
C07859=1016.836,177.790,375.549,167.477,53.174,159.875
C07860=1016.831,177.542,375.571,167.473,53.185,159.876
C07861=1016.826,177.293,375.591,167.469,53.195,159.878
C07862=1016.822,177.044,375.612,167.465,53.204,159.879
C07863=1016.817,176.794,375.633,167.461,53.214,159.880
C07864=1016.812,176.546,375.654,167.457,53.224,159.881
C07865=1016.807,176.296,375.676,167.452,53.234,159.882
C07866=1016.803,176.047,375.697,167.449,53.244,159.883
C07867=1016.797,175.798,375.717,167.445,53.254,159.885
C07868=1016.792,175.549,375.739,167.441,53.263,159.886
C07869=1016.788,175.301,375.759,167.437,53.273,159.887
C07870=1016.783,175.051,375.780,167.434,53.283,159.888
C07871=1016.779,174.802,375.802,167.428,53.293,159.889
C07872=1016.773,174.553,375.822,167.425,53.303,159.891
C07873=1016.769,174.304,375.844,167.421,53.312,159.892
C07874=1016.763,174.055,375.865,167.417,53.322,159.893
C07875=1016.759,173.806,375.885,167.414,53.332,159.894
C07876=1016.755,173.556,375.907,167.409,53.341,159.895
C07877=1016.750,173.307,375.927,167.406,53.351,159.896
C07878=1016.745,173.058,375.948,167.401,53.362,159.898
C07879=1016.740,172.809,375.969,167.397,53.371,159.899
C07880=1016.736,172.561,375.990,167.393,53.381,159.900
C07881=1016.731,172.311,376.011,167.390,53.391,159.901
C07882=1016.726,172.062,376.032,167.386,53.400,159.902
C07883=1016.721,171.813,376.053,167.382,53.410,159.904
C07884=1016.718,171.564,376.074,167.378,53.420,159.905
C07885=1016.712,171.283,376.097,167.374,53.431,159.906
C07886=1016.707,171.003,376.121,167.370,53.442,159.907
C07887=1016.701,170.722,376.144,167.366,53.453,159.909
C07888=1016.695,170.441,376.168,167.360,53.465,159.910
C07889=1016.692,170.192,376.188,167.356,53.474,159.911
C07890=1016.687,169.943,376.210,167.353,53.484,159.912
C07891=1016.681,169.694,376.231,167.349,53.494,159.914
C07892=1016.678,169.445,376.252,167.345,53.503,159.915
C07893=1016.672,169.196,376.272,167.341,53.513,159.916
C07894=1016.668,168.947,376.293,167.338,53.524,159.917
C07895=1016.664,168.698,376.314,167.334,53.533,159.918
C07896=1016.659,168.449,376.335,167.330,53.543,159.920
C07897=1016.654,168.199,376.356,167.326,53.552,159.921
C07898=1016.649,167.951,376.376,167.323,53.562,159.922
C07899=1016.645,167.702,376.397,167.319,53.572,159.923
C07900=1016.641,167.452,376.417,167.315,53.582,159.924
C07901=1016.636,167.203,376.438,167.311,53.592,159.926
C07902=1016.631,166.954,376.459,167.307,53.601,159.927
C07903=1016.626,166.705,376.479,167.304,53.611,159.928
C07904=1016.622,166.456,376.500,167.300,53.621,159.929
C07905=1016.618,166.206,376.521,167.296,53.631,159.930
C07906=1016.613,165.957,376.542,167.293,53.641,159.932
C07907=1016.609,165.709,376.563,167.289,53.650,159.933
C07908=1016.603,165.459,376.583,167.285,53.660,159.934
C07909=1016.599,165.211,376.604,167.281,53.670,159.935
C07910=1016.594,164.962,376.625,167.278,53.680,159.936
C07911=1016.590,164.712,376.646,167.274,53.690,159.938
C07912=1016.586,164.463,376.666,167.270,53.699,159.939
C07913=1016.581,164.214,376.686,167.266,53.709,159.940
C07914=1016.577,163.965,376.707,167.262,53.719,159.941
C07915=1016.572,163.716,376.728,167.259,53.729,159.942
C07916=1016.567,163.466,376.749,167.255,53.739,159.944
C07917=1016.563,163.218,376.770,167.251,53.748,159.945
C07918=1016.558,162.968,376.789,167.249,53.758,159.946
C07919=1016.554,162.719,376.810,167.245,53.767,159.947
C07920=1016.549,162.470,376.831,167.241,53.778,159.948
C07921=1016.545,162.221,376.851,167.237,53.787,159.950
C07922=1016.541,161.972,376.873,167.234,53.797,159.951
C07923=1016.536,161.723,376.892,167.230,53.806,159.952
C07924=1016.532,161.473,376.913,167.226,53.817,159.953
C07925=1016.527,161.225,376.933,167.223,53.827,159.954
C07926=1016.523,160.976,376.955,167.219,53.836,159.956
C07927=1016.518,160.726,376.974,167.215,53.846,159.957
C07928=1016.514,160.477,376.995,167.212,53.855,159.958
C07929=1016.510,160.228,377.016,167.209,53.865,159.959
C07930=1016.505,159.979,377.037,167.205,53.875,159.960
C07931=1016.501,159.730,377.057,167.201,53.885,159.962
C07932=1016.496,159.481,377.077,167.197,53.894,159.963
C07933=1016.492,159.232,377.098,167.194,53.904,159.964
C07934=1016.487,158.982,377.118,167.190,53.914,159.965
C07935=1016.483,158.733,377.139,167.186,53.924,159.966
C07936=1016.478,158.484,377.160,167.184,53.933,159.968
C07937=1016.474,158.235,377.179,167.180,53.943,159.969
C07938=1016.469,157.986,377.200,167.177,53.953,159.970
C07939=1016.464,157.737,377.219,167.173,53.964,159.971
C07940=1016.459,157.488,377.240,167.169,53.973,159.973
C07941=1016.455,157.239,377.259,167.166,53.983,159.974
C07942=1016.450,156.989,377.279,167.162,53.993,159.975
C07943=1016.445,156.741,377.299,167.159,54.003,159.976
C07944=1016.441,156.490,377.320,167.155,54.014,159.978
C07945=1016.436,156.242,377.340,167.151,54.023,159.979
C07946=1016.432,155.993,377.359,167.148,54.033,159.980
C07947=1016.427,155.743,377.379,167.144,54.043,159.981
C07948=1016.422,155.495,377.399,167.141,54.053,159.983
C07949=1016.417,155.213,377.422,167.137,54.065,159.984
C07950=1016.412,154.932,377.444,167.133,54.076,159.986
C07951=1016.407,154.652,377.467,167.129,54.087,159.987
C07952=1016.402,154.371,377.489,167.125,54.098,159.988
C07953=1016.397,154.122,377.509,167.121,54.108,159.989
C07954=1016.392,153.873,377.529,167.118,54.118,159.991
C07955=1016.387,153.623,377.549,167.114,54.128,159.992
C07956=1016.383,153.375,377.569,167.110,54.138,159.993
C07957=1016.378,153.126,377.588,167.107,54.148,159.994
C07958=1016.374,152.876,377.608,167.103,54.158,159.996
C07959=1016.370,152.626,377.628,167.100,54.168,159.997
C07960=1016.364,152.378,377.648,167.096,54.178,159.998
C07961=1016.360,152.129,377.668,167.094,54.188,159.999
C07962=1016.355,151.880,377.687,167.090,54.198,160.001
C07963=1016.350,151.630,377.707,167.087,54.208,160.002
C07964=1016.346,151.381,377.726,167.083,54.218,160.003
C07965=1016.341,151.131,377.746,167.080,54.228,160.005
C07966=1016.336,150.883,377.766,167.076,54.238,160.006
C07967=1016.332,150.634,377.786,167.073,54.248,160.007
C07968=1016.327,150.384,377.806,167.069,54.258,160.008
C07969=1016.323,150.135,377.825,167.066,54.268,160.010
C07970=1016.318,149.886,377.845,167.062,54.278,160.011
C07971=1016.313,149.636,377.865,167.058,54.288,160.012
C07972=1016.309,149.387,377.884,167.055,54.298,160.013
C07973=1016.305,149.138,377.904,167.052,54.308,160.015
C07974=1016.299,148.889,377.924,167.048,54.318,160.016
C07975=1016.295,148.640,377.944,167.045,54.328,160.017
C07976=1016.291,148.391,377.963,167.042,54.338,160.019
C07977=1016.286,148.142,377.982,167.039,54.348,160.020
C07978=1016.281,147.892,378.002,167.035,54.358,160.021
C07979=1016.276,147.643,378.021,167.031,54.368,160.022
C07980=1016.272,147.394,378.041,167.028,54.378,160.024
C07981=1016.267,147.144,378.061,167.025,54.388,160.025
C07982=1016.263,146.895,378.080,167.021,54.399,160.026
C07983=1016.258,146.646,378.099,167.017,54.408,160.027
C07984=1016.254,146.397,378.119,167.014,54.418,160.029
C07985=1016.249,146.147,378.139,167.012,54.428,160.030
C07986=1016.244,145.899,378.158,167.008,54.438,160.031
C07987=1016.240,145.650,378.177,167.005,54.449,160.033
C07988=1016.235,145.401,378.197,167.001,54.458,160.034
C07989=1016.230,145.151,378.216,166.998,54.468,160.035
C07990=1016.226,144.901,378.235,166.994,54.479,160.036
C07991=1016.221,144.653,378.254,166.991,54.489,160.038
C07992=1016.217,144.403,378.274,166.988,54.499,160.039
C07993=1016.212,144.154,378.293,166.984,54.509,160.040
C07994=1016.207,143.905,378.312,166.981,54.519,160.041
C07995=1016.202,143.656,378.332,166.977,54.529,160.043
C07996=1016.198,143.406,378.350,166.975,54.539,160.044
C07997=1016.193,143.157,378.370,166.972,54.549,160.045
C07998=1016.188,142.908,378.389,166.968,54.560,160.047
C07999=1016.184,142.659,378.409,166.965,54.570,160.048
C08000=1016.179,142.409,378.427,166.962,54.580,160.049
C08001=1016.175,142.160,378.446,166.958,54.590,160.050
C08002=1016.170,141.911,378.466,166.954,54.600,160.052
C08003=1016.165,141.662,378.485,166.951,54.610,160.053
C08004=1016.161,141.413,378.504,166.948,54.620,160.054
C08005=1016.156,141.163,378.523,166.946,54.630,160.056
C08006=1016.151,140.914,378.542,166.942,54.640,160.057
C08007=1016.146,140.665,378.562,166.938,54.650,160.058
C08008=1016.142,140.415,378.581,166.935,54.660,160.060
C08009=1016.137,140.166,378.600,166.932,54.671,160.061
C08010=1016.133,139.917,378.619,166.928,54.681,160.062
C08011=1016.129,139.668,378.639,166.925,54.690,160.063
C08012=1016.124,139.419,378.657,166.922,54.700,160.065
C08013=1016.119,139.138,378.679,166.919,54.712,160.066
C08014=1016.114,138.857,378.701,166.915,54.723,160.068
C08015=1016.108,138.576,378.721,166.911,54.734,160.069
C08016=1016.103,138.295,378.743,166.907,54.746,160.071
C08017=1016.099,138.046,378.763,166.905,54.756,160.072
C08018=1016.094,137.797,378.781,166.902,54.766,160.073
C08019=1016.089,137.547,378.801,166.898,54.776,160.075
C08020=1016.084,137.298,378.819,166.895,54.787,160.076
C08021=1016.080,137.048,378.838,166.891,54.796,160.077
C08022=1016.075,136.800,378.857,166.888,54.807,160.078
C08023=1016.071,136.550,378.876,166.885,54.817,160.080
C08024=1016.066,136.301,378.895,166.882,54.827,160.081
C08025=1016.062,136.052,378.914,166.879,54.837,160.083
C08026=1016.057,135.803,378.932,166.876,54.847,160.084
C08027=1016.053,135.553,378.951,166.872,54.857,160.085
C08028=1016.047,135.305,378.970,166.869,54.867,160.086
C08029=1016.043,135.054,378.989,166.866,54.878,160.088
C08030=1016.038,134.805,379.008,166.862,54.888,160.089
C08031=1016.033,134.556,379.026,166.860,54.898,160.090
C08032=1016.029,134.306,379.045,166.857,54.908,160.092
C08033=1016.024,134.058,379.064,166.854,54.918,160.093
C08034=1016.020,133.808,379.083,166.850,54.928,160.094
C08035=1016.015,133.559,379.101,166.847,54.938,160.095
C08036=1016.010,133.310,379.120,166.843,54.949,160.097
C08037=1016.006,133.060,379.138,166.840,54.959,160.098
C08038=1016.001,132.812,379.157,166.838,54.969,160.100
C08039=1015.997,132.562,379.176,166.835,54.979,160.101
C08040=1015.992,132.313,379.195,166.831,54.989,160.102
C08041=1015.987,132.064,379.213,166.828,54.999,160.103
C08042=1015.983,131.814,379.232,166.825,55.010,160.105
C08043=1015.978,131.565,379.251,166.822,55.019,160.106
C08044=1015.973,131.316,379.269,166.819,55.030,160.108
C08045=1015.969,131.066,379.288,166.815,55.039,160.109
C08046=1015.964,130.818,379.306,166.812,55.050,160.110
C08047=1015.960,130.568,379.325,166.809,55.060,160.111
C08048=1015.955,130.319,379.343,166.807,55.070,160.113
C08049=1015.950,130.070,379.362,166.804,55.080,160.114
C08050=1015.946,129.820,379.381,166.800,55.090,160.115
C08051=1015.941,129.571,379.399,166.797,55.100,160.117
C08052=1015.936,129.322,379.417,166.794,55.111,160.118
C08053=1015.931,129.073,379.436,166.791,55.121,160.119
C08054=1015.927,128.823,379.455,166.788,55.131,160.121
C08055=1015.922,128.574,379.473,166.785,55.141,160.122
C08056=1015.918,128.325,379.491,166.782,55.152,160.123
C08057=1015.913,128.075,379.509,166.779,55.162,160.125
C08058=1015.908,127.826,379.528,166.775,55.173,160.126
C08059=1015.903,127.576,379.546,166.772,55.183,160.127
C08060=1015.899,127.327,379.564,166.769,55.193,160.129
C08061=1015.894,127.078,379.582,166.766,55.204,160.130
C08062=1015.889,126.828,379.600,166.764,55.214,160.132
C08063=1015.884,126.579,379.618,166.761,55.224,160.133
C08064=1015.879,126.330,379.637,166.757,55.234,160.134
C08065=1015.874,126.081,379.655,166.754,55.244,160.135
C08066=1015.870,125.832,379.674,166.751,55.254,160.137
C08067=1015.865,125.582,379.692,166.748,55.265,160.138
C08068=1015.860,125.333,379.710,166.744,55.275,160.139
C08069=1015.855,125.084,379.728,166.742,55.285,160.141
C08070=1015.850,124.834,379.746,166.739,55.295,160.142
C08071=1015.846,124.585,379.764,166.736,55.306,160.144
C08072=1015.841,124.336,379.782,166.733,55.316,160.145
C08073=1015.837,124.087,379.800,166.730,55.327,160.146
C08074=1015.832,123.838,379.819,166.726,55.336,160.147
C08075=1015.827,123.588,379.837,166.724,55.346,160.149
C08076=1015.822,123.339,379.855,166.721,55.357,160.150
C08077=1015.817,123.058,379.876,166.717,55.368,160.152
C08078=1015.812,122.777,379.895,166.713,55.380,160.153
C08079=1015.807,122.495,379.916,166.710,55.391,160.155
C08080=1015.801,122.214,379.936,166.708,55.403,160.157
C08081=1015.797,121.965,379.954,166.704,55.413,160.158
C08082=1015.792,121.716,379.972,166.701,55.423,160.159
C08083=1015.788,121.467,379.990,166.698,55.434,160.160
C08084=1015.783,121.217,380.009,166.696,55.444,160.162
C08085=1015.778,120.968,380.027,166.693,55.454,160.163
C08086=1015.773,120.719,380.045,166.689,55.464,160.164
C08087=1015.768,120.469,380.063,166.686,55.474,160.166
C08088=1015.764,120.221,380.081,166.684,55.484,160.167
C08089=1015.759,119.971,380.099,166.681,55.495,160.169
C08090=1015.755,119.721,380.116,166.678,55.505,160.170
C08091=1015.750,119.472,380.135,166.674,55.515,160.171
C08092=1015.745,119.223,380.153,166.672,55.525,160.173
C08093=1015.741,118.973,380.171,166.669,55.535,160.174
C08094=1015.736,118.725,380.189,166.666,55.546,160.175
C08095=1015.732,118.475,380.207,166.663,55.556,160.177
C08096=1015.727,118.226,380.225,166.660,55.565,160.178
C08097=1015.722,117.976,380.243,166.657,55.576,160.179
C08098=1015.718,117.726,380.261,166.654,55.586,160.181
C08099=1015.714,117.478,380.279,166.651,55.596,160.182
C08100=1015.709,117.228,380.297,166.648,55.606,160.183
C08101=1015.705,116.979,380.315,166.645,55.616,160.185
C08102=1015.700,116.730,380.334,166.643,55.626,160.186
C08103=1015.696,116.480,380.351,166.640,55.636,160.187
C08104=1015.691,116.231,380.369,166.637,55.647,160.189
C08105=1015.686,115.982,380.387,166.634,55.657,160.190
C08106=1015.682,115.732,380.405,166.631,55.666,160.191
C08107=1015.677,115.484,380.423,166.628,55.677,160.193
C08108=1015.673,115.234,380.440,166.625,55.687,160.194
C08109=1015.668,114.984,380.459,166.622,55.697,160.195
C08110=1015.663,114.735,380.477,166.619,55.707,160.197
C08111=1015.659,114.486,380.495,166.617,55.717,160.198
C08112=1015.655,114.236,380.512,166.614,55.727,160.199
C08113=1015.650,113.987,380.530,166.611,55.737,160.201
C08114=1015.645,113.738,380.548,166.609,55.747,160.202
C08115=1015.641,113.489,380.566,166.605,55.757,160.203
C08116=1015.637,113.239,380.584,166.602,55.768,160.205
C08117=1015.632,112.990,380.602,166.600,55.778,160.206
C08118=1015.628,112.741,380.619,166.597,55.787,160.207
C08119=1015.623,112.492,380.638,166.595,55.797,160.209
C08120=1015.618,112.242,380.655,166.591,55.807,160.210
C08121=1015.614,111.992,380.673,166.588,55.818,160.211
C08122=1015.609,111.744,380.691,166.586,55.828,160.213
C08123=1015.604,111.494,380.708,166.583,55.838,160.214
C08124=1015.599,111.245,380.726,166.580,55.848,160.215
C08125=1015.596,110.995,380.743,166.577,55.859,160.217
C08126=1015.590,110.746,380.761,166.575,55.869,160.218
C08127=1015.586,110.496,380.778,166.572,55.879,160.219
C08128=1015.581,110.247,380.796,166.568,55.889,160.221
C08129=1015.577,109.998,380.813,166.566,55.899,160.222
C08130=1015.571,109.749,380.831,166.563,55.909,160.224
C08131=1015.567,109.499,380.848,166.560,55.920,160.225
C08132=1015.563,109.250,380.866,166.558,55.929,160.226
C08133=1015.557,109.001,380.883,166.555,55.940,160.228
C08134=1015.553,108.751,380.901,166.552,55.950,160.229
C08135=1015.548,108.502,380.918,166.549,55.961,160.230
C08136=1015.544,108.252,380.935,166.547,55.971,160.232
C08137=1015.539,108.003,380.953,166.543,55.981,160.233
C08138=1015.534,107.754,380.970,166.540,55.991,160.234
C08139=1015.530,107.504,380.987,166.537,56.002,160.236
C08140=1015.524,107.255,381.005,166.535,56.012,160.237
C08141=1015.517,106.847,381.033,166.531,56.029,160.239
C08142=1015.509,106.439,381.061,166.526,56.046,160.242
C08143=1015.502,106.030,381.089,166.522,56.062,160.244
C08144=1015.494,105.622,381.117,166.517,56.079,160.246
C08145=1015.487,105.250,381.144,166.513,56.094,160.248
C08146=1015.480,104.879,381.169,166.508,56.109,160.250
C08147=1015.473,104.508,381.194,166.505,56.124,160.252
C08148=1015.467,104.137,381.220,166.500,56.140,160.254
C08149=1015.461,103.887,381.238,166.498,56.149,160.256
C08150=1015.457,103.637,381.255,166.495,56.160,160.257
C08151=1015.452,103.389,381.272,166.493,56.170,160.259
C08152=1015.447,103.139,381.289,166.489,56.180,160.260
C08153=1015.443,102.890,381.306,166.487,56.190,160.261
C08154=1015.438,102.640,381.324,166.485,56.200,160.263
C08155=1015.433,102.391,381.340,166.481,56.210,160.264
C08156=1015.429,102.141,381.358,166.478,56.221,160.265
C08157=1015.424,101.893,381.375,166.476,56.231,160.267
C08158=1015.420,101.643,381.392,166.473,56.241,160.268
C08159=1015.414,101.393,381.409,166.470,56.251,160.269
C08160=1015.411,101.144,381.426,166.468,56.261,160.271
C08161=1015.405,100.894,381.443,166.465,56.271,160.272
C08162=1015.401,100.646,381.461,166.463,56.281,160.273
C08163=1015.396,100.396,381.478,166.460,56.291,160.275
C08164=1015.392,100.147,381.495,166.457,56.302,160.276
C08165=1015.388,99.897,381.512,166.455,56.312,160.278
C08166=1015.383,99.648,381.529,166.451,56.322,160.279
C08167=1015.378,99.399,381.547,166.450,56.332,160.280
C08168=1015.374,99.150,381.563,166.446,56.342,160.281
C08169=1015.369,98.900,381.581,166.444,56.352,160.283
C08170=1015.364,98.651,381.597,166.441,56.363,160.284
C08171=1015.359,98.401,381.614,166.438,56.372,160.285
C08172=1015.355,98.152,381.631,166.435,56.383,160.287
C08173=1015.350,97.902,381.648,166.433,56.393,160.288
C08174=1015.346,97.653,381.664,166.430,56.403,160.290
C08175=1015.340,97.403,381.681,166.427,56.414,160.291
C08176=1015.336,97.155,381.698,166.425,56.424,160.293
C08177=1015.331,96.905,381.715,166.422,56.434,160.294
C08178=1015.327,96.656,381.732,166.419,56.444,160.295
C08179=1015.321,96.406,381.749,166.417,56.454,160.297
C08180=1015.317,96.157,381.765,166.414,56.465,160.298
C08181=1015.312,95.907,381.781,166.412,56.474,160.299
C08182=1015.307,95.658,381.798,166.409,56.485,160.301
C08183=1015.303,95.408,381.815,166.406,56.496,160.302
C08184=1015.298,95.159,381.832,166.404,56.505,160.303
C08185=1015.293,94.909,381.848,166.401,56.516,160.305
C08186=1015.288,94.660,381.865,166.398,56.525,160.306
C08187=1015.284,94.410,381.882,166.396,56.536,160.308
C08188=1015.279,94.161,381.899,166.393,56.546,160.309
C08189=1015.275,93.912,381.915,166.391,56.556,160.310
C08190=1015.270,93.663,381.932,166.388,56.566,160.312
C08191=1015.265,93.414,381.949,166.385,56.576,160.313
C08192=1015.261,93.163,381.965,166.383,56.586,160.314
C08193=1015.256,92.914,381.982,166.380,56.597,160.316
C08194=1015.251,92.664,381.999,166.378,56.606,160.317
C08195=1015.246,92.416,382.015,166.375,56.617,160.319
C08196=1015.242,92.167,382.032,166.372,56.627,160.320
C08197=1015.237,91.917,382.049,166.370,56.637,160.321
C08198=1015.233,91.668,382.066,166.366,56.647,160.322
C08199=1015.227,91.418,382.083,166.365,56.657,160.324
C08200=1015.223,91.168,382.098,166.361,56.667,160.325
C08201=1015.218,90.888,382.117,166.359,56.678,160.327
C08202=1015.212,90.607,382.136,166.356,56.690,160.328
C08203=1015.208,90.327,382.155,166.353,56.701,160.330
C08204=1015.202,90.046,382.174,166.350,56.713,160.331
C08205=1015.198,89.797,382.190,166.348,56.723,160.333
C08206=1015.193,89.547,382.206,166.345,56.733,160.334
C08207=1015.189,89.297,382.223,166.342,56.742,160.335
C08208=1015.184,89.048,382.240,166.340,56.753,160.337
C08209=1015.179,88.799,382.257,166.337,56.762,160.338
C08210=1015.175,88.549,382.273,166.335,56.773,160.340
C08211=1015.170,88.300,382.289,166.332,56.784,160.341
C08212=1015.165,88.051,382.306,166.330,56.793,160.342
C08213=1015.161,87.801,382.322,166.327,56.804,160.344
C08214=1015.156,87.551,382.339,166.325,56.813,160.345
C08215=1015.150,87.302,382.354,166.322,56.824,160.346
C08216=1015.145,87.052,382.371,166.319,56.835,160.348
C08217=1015.141,86.803,382.387,166.317,56.844,160.349
C08218=1015.136,86.554,382.403,166.314,56.855,160.351
C08219=1015.131,86.304,382.420,166.311,56.865,160.352
C08220=1015.127,86.055,382.435,166.309,56.875,160.353
C08221=1015.122,85.806,382.452,166.306,56.885,160.355
C08222=1015.118,85.556,382.468,166.304,56.895,160.356
C08223=1015.113,85.306,382.485,166.301,56.906,160.358
C08224=1015.108,85.058,382.501,166.299,56.915,160.359
C08225=1015.103,84.808,382.516,166.296,56.926,160.360
C08226=1015.098,84.559,382.533,166.293,56.936,160.362
C08227=1015.094,84.309,382.549,166.291,56.946,160.363
C08228=1015.089,84.060,382.565,166.288,56.956,160.364
C08229=1015.084,83.810,382.581,166.287,56.966,160.366
C08230=1015.079,83.561,382.598,166.283,56.976,160.367
C08231=1015.075,83.311,382.614,166.282,56.986,160.369
C08232=1015.070,83.062,382.631,166.278,56.996,160.370
C08233=1015.066,82.812,382.646,166.276,57.006,160.371
C08234=1015.060,82.563,382.662,166.273,57.017,160.373
C08235=1015.056,82.314,382.678,166.271,57.026,160.374
C08236=1015.051,82.064,382.695,166.269,57.037,160.375
C08237=1015.046,81.815,382.711,166.266,57.046,160.377
C08238=1015.042,81.566,382.727,166.264,57.057,160.378
C08239=1015.037,81.316,382.743,166.260,57.067,160.379
C08240=1015.032,81.066,382.760,166.258,57.077,160.381
C08241=1015.028,80.817,382.775,166.257,57.087,160.382
C08242=1015.023,80.567,382.791,166.253,57.097,160.383
C08243=1015.018,80.319,382.807,166.251,57.106,160.385
C08244=1015.013,80.068,382.823,166.248,57.117,160.386
C08245=1015.009,79.819,382.840,166.246,57.127,160.388
C08246=1015.004,79.570,382.856,166.243,57.136,160.389
C08247=1015.000,79.321,382.872,166.241,57.147,160.390
C08248=1014.995,79.070,382.888,166.238,57.157,160.391
C08249=1014.991,78.821,382.904,166.236,57.166,160.393
C08250=1014.986,78.572,382.920,166.233,57.177,160.394
C08251=1014.981,78.323,382.936,166.231,57.187,160.396
C08252=1014.976,78.074,382.952,166.228,57.197,160.397
C08253=1014.971,77.823,382.968,166.226,57.207,160.398
C08254=1014.967,77.574,382.984,166.224,57.216,160.400
C08255=1014.963,77.325,383.000,166.221,57.226,160.401
C08256=1014.958,77.075,383.016,166.219,57.236,160.402
C08257=1014.954,76.826,383.032,166.216,57.247,160.404
C08258=1014.948,76.576,383.048,166.214,57.256,160.405
C08259=1014.944,76.327,383.064,166.211,57.266,160.406
C08260=1014.939,76.077,383.080,166.209,57.276,160.408
C08261=1014.934,75.828,383.095,166.206,57.286,160.409
C08262=1014.930,75.579,383.111,166.204,57.296,160.410
C08263=1014.925,75.329,383.127,166.201,57.307,160.412
C08264=1014.920,75.079,383.143,166.199,57.316,160.413
C08265=1014.915,74.799,383.160,166.197,57.328,160.415
C08266=1014.910,74.519,383.179,166.193,57.339,160.416
C08267=1014.904,74.238,383.196,166.191,57.350,160.418
C08268=1014.899,73.957,383.214,166.188,57.362,160.419
C08269=1014.894,73.708,383.229,166.186,57.371,160.421
C08270=1014.890,73.459,383.244,166.183,57.382,160.422
C08271=1014.885,73.210,383.261,166.181,57.391,160.423
C08272=1014.879,72.960,383.276,166.178,57.401,160.425
C08273=1014.875,72.710,383.292,166.176,57.412,160.426
C08274=1014.870,72.461,383.307,166.174,57.421,160.428
C08275=1014.866,72.211,383.323,166.171,57.431,160.429
C08276=1014.861,71.962,383.339,166.169,57.441,160.430
C08277=1014.856,71.712,383.354,166.166,57.452,160.432
C08278=1014.852,71.463,383.370,166.164,57.461,160.433
C08279=1014.847,71.214,383.385,166.161,57.471,160.434
C08280=1014.842,70.964,383.402,166.159,57.481,160.435
C08281=1014.837,70.715,383.417,166.157,57.491,160.437
C08282=1014.832,70.465,383.433,166.154,57.501,160.438
C08283=1014.828,70.215,383.449,166.152,57.511,160.440
C08284=1014.823,69.966,383.464,166.149,57.521,160.441
C08285=1014.819,69.717,383.480,166.147,57.531,160.442
C08286=1014.814,69.467,383.495,166.144,57.541,160.443
C08287=1014.809,69.218,383.511,166.142,57.551,160.445
C08288=1014.804,68.969,383.526,166.140,57.560,160.446
C08289=1014.800,68.719,383.541,166.137,57.571,160.448
C08290=1014.795,68.470,383.557,166.135,57.580,160.449
C08291=1014.791,68.220,383.572,166.133,57.590,160.450
C08292=1014.785,67.970,383.588,166.130,57.600,160.451
C08293=1014.781,67.721,383.604,166.128,57.610,160.453
C08294=1014.776,67.471,383.619,166.125,57.620,160.454
C08295=1014.771,67.222,383.635,166.123,57.630,160.456
C08296=1014.766,66.972,383.650,166.121,57.639,160.457
C08297=1014.761,66.723,383.665,166.118,57.649,160.458
C08298=1014.757,66.474,383.681,166.116,57.659,160.460
C08299=1014.752,66.224,383.695,166.113,57.670,160.461
C08300=1014.748,65.974,383.711,166.111,57.679,160.462
C08301=1014.743,65.725,383.726,166.109,57.689,160.464
C08302=1014.738,65.476,383.741,166.106,57.699,160.465
C08303=1014.734,65.226,383.757,166.104,57.709,160.466
C08304=1014.729,64.977,383.772,166.101,57.719,160.468
C08305=1014.724,64.727,383.788,166.099,57.728,160.469
C08306=1014.720,64.477,383.803,166.097,57.739,160.471
C08307=1014.715,64.228,383.818,166.094,57.749,160.472
C08308=1014.710,63.978,383.833,166.092,57.759,160.473
C08309=1014.705,63.729,383.849,166.090,57.768,160.475
C08310=1014.700,63.480,383.864,166.087,57.778,160.476
C08311=1014.696,63.230,383.880,166.085,57.788,160.477
C08312=1014.691,62.980,383.894,166.082,57.798,160.478
C08313=1014.686,62.731,383.909,166.080,57.808,160.480
C08314=1014.682,62.482,383.925,166.078,57.817,160.481
C08315=1014.677,62.232,383.939,166.075,57.827,160.482
C08316=1014.672,61.982,383.955,166.074,57.838,160.484
C08317=1014.667,61.733,383.970,166.071,57.848,160.485
C08318=1014.662,61.483,383.984,166.069,57.857,160.487
C08319=1014.657,61.234,383.999,166.065,57.868,160.488
C08320=1014.652,60.984,384.014,166.063,57.877,160.489
C08321=1014.647,60.735,384.029,166.062,57.888,160.491
C08322=1014.642,60.486,384.044,166.059,57.898,160.492
C08323=1014.638,60.236,384.059,166.057,57.907,160.493
C08324=1014.633,59.986,384.074,166.054,57.917,160.495
C08325=1014.628,59.737,384.088,166.052,57.927,160.496
C08326=1014.623,59.487,384.104,166.049,57.937,160.497
C08327=1014.618,59.237,384.118,166.047,57.947,160.499
C08328=1014.613,58.988,384.133,166.045,57.956,160.500
C08329=1014.607,58.708,384.150,166.042,57.968,160.502
C08330=1014.602,58.427,384.166,166.040,57.979,160.503
C08331=1014.596,58.147,384.183,166.037,57.990,160.505
C08332=1014.591,57.866,384.200,166.034,58.001,160.506
C08333=1014.586,57.617,384.215,166.032,58.011,160.507
C08334=1014.581,57.367,384.230,166.030,58.021,160.509
C08335=1014.577,57.118,384.244,166.027,58.031,160.510
C08336=1014.572,56.869,384.259,166.025,58.041,160.511
C08337=1014.567,56.619,384.274,166.023,58.050,160.513
C08338=1014.562,56.370,384.289,166.020,58.060,160.514
C08339=1014.558,56.120,384.303,166.018,58.070,160.515
C08340=1014.553,55.871,384.319,166.016,58.080,160.517
C08341=1014.548,55.621,384.333,166.013,58.090,160.518
C08342=1014.543,55.371,384.347,166.011,58.099,160.519
C08343=1014.538,55.122,384.363,166.009,58.109,160.521
C08344=1014.534,54.872,384.377,166.006,58.119,160.522
C08345=1014.529,54.623,384.392,166.004,58.129,160.523
C08346=1014.524,54.373,384.406,166.002,58.139,160.525
C08347=1014.519,54.124,384.422,166.000,58.148,160.526
C08348=1014.514,53.874,384.436,165.997,58.158,160.527
C08349=1014.509,53.625,384.451,165.995,58.168,160.529
C08350=1014.505,53.375,384.466,165.993,58.177,160.530
C08351=1014.500,53.126,384.480,165.990,58.187,160.531
C08352=1014.495,52.877,384.495,165.988,58.197,160.532
C08353=1014.491,52.627,384.509,165.986,58.207,160.534
C08354=1014.486,52.377,384.525,165.984,58.216,160.535
C08355=1014.481,52.127,384.539,165.980,58.226,160.536
C08356=1014.476,51.878,384.554,165.979,58.235,160.538
C08357=1014.472,51.629,384.568,165.977,58.245,160.539
C08358=1014.467,51.379,384.583,165.975,58.255,160.540
C08359=1014.462,51.130,384.598,165.973,58.265,160.542
C08360=1014.457,50.880,384.612,165.969,58.274,160.543
C08361=1014.452,50.631,384.628,165.967,58.284,160.544
C08362=1014.447,50.381,384.642,165.965,58.293,160.546
C08363=1014.443,50.132,384.656,165.963,58.302,160.547
C08364=1014.438,49.882,384.671,165.961,58.312,160.548
C08365=1014.434,49.633,384.686,165.959,58.322,160.550
C08366=1014.429,49.383,384.700,165.956,58.332,160.551
C08367=1014.424,49.133,384.715,165.954,58.341,160.552
C08368=1014.420,48.884,384.729,165.952,58.351,160.553
C08369=1014.415,48.634,384.744,165.950,58.360,160.555
C08370=1014.410,48.385,384.759,165.947,58.369,160.556
C08371=1014.405,48.135,384.774,165.946,58.379,160.557
C08372=1014.401,47.886,384.788,165.942,58.389,160.558
C08373=1014.396,47.637,384.803,165.940,58.398,160.560
C08374=1014.391,47.387,384.817,165.938,58.408,160.561
C08375=1014.386,47.137,384.832,165.936,58.417,160.562
C08376=1014.382,46.888,384.847,165.934,58.427,160.563
C08377=1014.377,46.638,384.861,165.931,58.436,160.565
C08378=1014.373,46.389,384.875,165.930,58.445,160.566
C08379=1014.367,46.139,384.891,165.927,58.454,160.567
C08380=1014.364,45.890,384.905,165.925,58.464,160.569
C08381=1014.359,45.640,384.920,165.923,58.473,160.570
C08382=1014.355,45.390,384.934,165.921,58.483,160.571
C08383=1014.350,45.141,384.949,165.918,58.492,160.572
C08384=1014.345,44.892,384.963,165.916,58.502,160.573
C08385=1014.341,44.642,384.978,165.913,58.511,160.575
C08386=1014.336,44.392,384.992,165.911,58.521,160.576
C08387=1014.331,44.143,385.008,165.909,58.530,160.577
C08388=1014.327,43.893,385.022,165.907,58.540,160.578
C08389=1014.322,43.643,385.036,165.905,58.549,160.580
C08390=1014.317,43.394,385.051,165.902,58.558,160.581
C08391=1014.313,43.145,385.065,165.900,58.567,160.582
C08392=1014.308,42.895,385.080,165.898,58.576,160.583
C08393=1014.303,42.614,385.096,165.896,58.586,160.585
C08394=1014.297,42.334,385.112,165.894,58.597,160.586
C08395=1014.292,42.054,385.129,165.891,58.607,160.587
C08396=1014.287,41.773,385.145,165.889,58.618,160.589
C08397=1014.282,41.523,385.159,165.886,58.627,160.590
C08398=1014.277,41.275,385.173,165.884,58.637,160.592
C08399=1014.272,41.025,385.187,165.882,58.646,160.593
C08400=1014.268,40.775,385.202,165.880,58.656,160.594
C08401=1014.264,40.526,385.216,165.877,58.665,160.595
C08402=1014.258,40.276,385.229,165.875,58.675,160.597
C08403=1014.253,40.026,385.244,165.872,58.684,160.598
C08404=1014.249,39.777,385.258,165.870,58.693,160.599
C08405=1014.244,39.527,385.272,165.868,58.703,160.600
C08406=1014.239,39.277,385.286,165.866,58.712,160.601
C08407=1014.235,39.028,385.300,165.864,58.722,160.603
C08408=1014.229,38.779,385.314,165.862,58.731,160.604
C08409=1014.225,38.530,385.328,165.859,58.740,160.605
C08410=1014.221,38.280,385.343,165.857,58.749,160.606
C08411=1014.216,38.030,385.357,165.855,58.758,160.608
C08412=1014.211,37.781,385.371,165.853,58.767,160.609
C08413=1014.206,37.531,385.385,165.851,58.777,160.610
C08414=1014.201,37.281,385.400,165.848,58.786,160.611
C08415=1014.197,37.032,385.413,165.846,58.795,160.612
C08416=1014.192,36.782,385.427,165.844,58.805,160.614
C08417=1014.188,36.533,385.441,165.842,58.814,160.615
C08418=1014.183,36.283,385.456,165.839,58.823,160.616
C08419=1014.178,36.033,385.469,165.837,58.832,160.617
C08420=1014.174,35.784,385.483,165.835,58.842,160.619
C08421=1014.168,35.534,385.497,165.833,58.851,160.620
C08422=1014.164,35.285,385.510,165.831,58.861,160.621
C08423=1014.159,35.035,385.525,165.829,58.870,160.622
C08424=1014.153,34.785,385.538,165.826,58.879,160.624
C08425=1014.149,34.536,385.553,165.825,58.889,160.625
C08426=1014.144,34.286,385.566,165.822,58.898,160.626
C08427=1014.140,34.037,385.580,165.820,58.907,160.627
C08428=1014.134,33.787,385.594,165.818,58.916,160.628
C08429=1014.130,33.538,385.608,165.816,58.926,160.630
C08430=1014.125,33.288,385.621,165.813,58.935,160.631
C08431=1014.120,33.038,385.635,165.811,58.944,160.632
C08432=1014.116,32.789,385.649,165.809,58.953,160.633
C08433=1014.110,32.539,385.662,165.807,58.963,160.635
C08434=1014.106,32.290,385.676,165.805,58.972,160.636
C08435=1014.101,32.040,385.690,165.802,58.981,160.637
C08436=1014.097,31.791,385.704,165.800,58.990,160.638
C08437=1014.091,31.541,385.717,165.798,58.999,160.639
C08438=1014.087,31.292,385.731,165.796,59.009,160.641
C08439=1014.082,31.042,385.745,165.795,59.017,160.642
C08440=1014.078,30.792,385.759,165.792,59.026,160.643
C08441=1014.073,30.543,385.772,165.790,59.036,160.644
C08442=1014.068,30.294,385.786,165.787,59.045,160.646
C08443=1014.063,30.043,385.800,165.785,59.054,160.647
C08444=1014.058,29.794,385.813,165.783,59.063,160.648
C08445=1014.054,29.545,385.828,165.780,59.072,160.649
C08446=1014.049,29.295,385.840,165.778,59.081,160.650
C08447=1014.044,29.045,385.855,165.776,59.090,160.651
C08448=1014.039,28.796,385.868,165.775,59.099,160.653
C08449=1014.035,28.546,385.882,165.772,59.108,160.654
C08450=1014.030,28.297,385.896,165.770,59.117,160.655
C08451=1014.025,28.047,385.909,165.768,59.126,160.656
C08452=1014.021,27.797,385.923,165.765,59.135,160.657
C08453=1014.015,27.548,385.937,165.763,59.144,160.658
C08454=1014.012,27.298,385.950,165.762,59.153,160.660
C08455=1014.006,27.049,385.964,165.759,59.162,160.661
C08456=1014.001,26.799,385.977,165.757,59.171,160.662
C08457=1013.996,26.519,385.992,165.754,59.181,160.663
C08458=1013.990,26.238,386.007,165.752,59.191,160.664
C08459=1013.985,25.958,386.023,165.750,59.201,160.666
C08460=1013.980,25.678,386.038,165.747,59.212,160.667
C08461=1013.975,25.428,386.051,165.745,59.221,160.668
C08462=1013.970,25.179,386.065,165.743,59.230,160.670
C08463=1013.965,24.929,386.078,165.741,59.238,160.671
C08464=1013.961,24.679,386.091,165.739,59.247,160.672
C08465=1013.957,24.430,386.105,165.737,59.257,160.673
C08466=1013.951,24.180,386.118,165.734,59.266,160.674
C08467=1013.947,23.931,386.131,165.732,59.275,160.676
C08468=1013.941,23.681,386.145,165.730,59.284,160.677
C08469=1013.937,23.431,386.157,165.729,59.293,160.678
C08470=1013.933,23.182,386.172,165.726,59.302,160.679
C08471=1013.927,22.932,386.185,165.724,59.311,160.680
C08472=1013.923,22.683,386.198,165.721,59.319,160.681
C08473=1013.917,22.433,386.211,165.719,59.328,160.682
C08474=1013.913,22.183,386.224,165.718,59.337,160.684
C08475=1013.909,21.934,386.238,165.715,59.346,160.685
C08476=1013.904,21.684,386.251,165.713,59.355,160.686
C08477=1013.899,21.435,386.264,165.710,59.364,160.687
C08478=1013.894,21.185,386.278,165.709,59.372,160.688
C08479=1013.889,20.935,386.291,165.707,59.381,160.689
C08480=1013.884,20.686,386.304,165.704,59.390,160.691
C08481=1013.880,20.436,386.318,165.703,59.398,160.692
C08482=1013.875,20.187,386.331,165.700,59.407,160.693
C08483=1013.871,19.937,386.344,165.698,59.417,160.694
C08484=1013.865,19.688,386.357,165.696,59.426,160.695
C08485=1013.860,19.438,386.370,165.694,59.434,160.696
C08486=1013.857,19.188,386.384,165.692,59.443,160.697
C08487=1013.851,18.938,386.397,165.689,59.452,160.698
C08488=1013.847,18.689,386.410,165.688,59.460,160.699
C08489=1013.841,18.439,386.423,165.685,59.469,160.701
C08490=1013.837,18.189,386.436,165.683,59.478,160.702
C08491=1013.832,17.940,386.449,165.681,59.486,160.703
C08492=1013.827,17.691,386.462,165.679,59.495,160.704
C08493=1013.822,17.441,386.476,165.677,59.504,160.705
C08494=1013.818,17.191,386.488,165.675,59.512,160.706
C08495=1013.813,16.942,386.501,165.673,59.521,160.707
C08496=1013.808,16.692,386.514,165.671,59.531,160.709
C08497=1013.803,16.442,386.527,165.669,59.538,160.710
C08498=1013.798,16.193,386.541,165.666,59.548,160.711
C08499=1013.793,15.943,386.554,165.664,59.556,160.712
C08500=1013.789,15.694,386.567,165.662,59.565,160.713
C08501=1013.785,15.444,386.580,165.660,59.573,160.714
C08502=1013.780,15.194,386.593,165.657,59.582,160.715
C08503=1013.775,14.944,386.606,165.656,59.590,160.716
C08504=1013.771,14.695,386.619,165.653,59.599,160.717
C08505=1013.766,14.445,386.631,165.651,59.607,160.718
C08506=1013.761,14.196,386.645,165.649,59.616,160.719
C08507=1013.756,13.946,386.658,165.646,59.625,160.720
C08508=1013.751,13.697,386.671,165.645,59.634,160.722
C08509=1013.747,13.447,386.684,165.642,59.642,160.722
C08510=1013.742,13.197,386.697,165.641,59.651,160.724
C08511=1013.737,12.947,386.710,165.638,59.659,160.725
C08512=1013.733,12.698,386.722,165.637,59.668,160.726
C08513=1013.727,12.448,386.735,165.634,59.676,160.727
C08514=1013.722,12.199,386.748,165.632,59.685,160.728
C08515=1013.717,11.949,386.760,165.630,59.693,160.729
C08516=1013.713,11.699,386.773,165.628,59.702,160.730
C08517=1013.708,11.450,386.785,165.625,59.711,160.731
C08518=1013.703,11.200,386.798,165.624,59.720,160.733
C08519=1013.698,10.950,386.811,165.621,59.728,160.733
C08520=1013.694,10.701,386.823,165.620,59.737,160.735
C08521=1013.688,10.422,386.837,165.617,59.746,160.736
C08522=1013.682,10.143,386.851,165.615,59.755,160.737
C08523=1013.677,9.864,386.865,165.613,59.765,160.739
C08524=1013.672,9.586,386.879,165.610,59.775,160.739
C08525=1013.667,9.336,386.892,165.608,59.783,160.741
C08526=1013.662,9.086,386.905,165.605,59.791,160.741
C08527=1013.657,8.837,386.917,165.604,59.800,160.743
C08528=1013.652,8.587,386.930,165.601,59.809,160.744
C08529=1013.648,8.337,386.942,165.600,59.817,160.745
C08530=1013.643,8.088,386.955,165.598,59.826,160.746
C08531=1013.637,7.838,386.967,165.596,59.834,160.747
C08532=1013.633,7.588,386.980,165.593,59.842,160.748
C08533=1013.628,7.339,386.993,165.592,59.851,160.749
C08534=1013.624,7.089,387.005,165.589,59.859,160.750
C08535=1013.619,6.840,387.017,165.587,59.867,160.751
C08536=1013.614,6.590,387.030,165.584,59.876,160.752
C08537=1013.610,6.341,387.043,165.583,59.884,160.753
C08538=1013.604,6.090,387.056,165.581,59.893,160.754
C08539=1013.599,5.841,387.067,165.579,59.901,160.755
C08540=1013.595,5.591,387.080,165.577,59.909,160.756
C08541=1013.590,5.342,387.093,165.574,59.917,160.757
C08542=1013.585,5.092,387.105,165.572,59.925,160.758
C08543=1013.581,4.842,387.117,165.570,59.934,160.759
C08544=1013.576,4.593,387.130,165.568,59.942,160.760
C08545=1013.572,4.343,387.143,165.566,59.950,160.761
C08546=1013.566,4.093,387.155,165.563,59.958,160.762
C08547=1013.561,3.843,387.167,165.562,59.966,160.763
C08548=1013.557,3.594,387.180,165.560,59.974,160.764
C08549=1013.552,3.344,387.193,165.557,59.983,160.765
C08550=1013.547,3.095,387.205,165.555,59.991,160.766
C08551=1013.543,2.845,387.217,165.554,59.999,160.767
C08552=1013.538,2.596,387.230,165.551,60.007,160.768
C08553=1013.534,2.346,387.243,165.549,60.015,160.769
C08554=1013.529,2.096,387.254,165.547,60.023,160.770
C08555=1013.524,1.847,387.267,165.545,60.031,160.771
C08556=1013.519,1.597,387.280,165.543,60.039,160.772
C08557=1013.514,1.348,387.292,165.541,60.047,160.773
C08558=1013.509,1.097,387.304,165.539,60.055,160.774
C08559=1013.505,0.848,387.317,165.537,60.064,160.775
C08560=1013.500,0.598,387.330,165.534,60.071,160.776
C08561=1013.495,0.349,387.341,165.533,60.079,160.777
C08562=1013.491,0.099,387.354,165.531,60.087,160.778
C08563=1013.486,-0.150,387.367,165.528,60.096,160.779
C08564=1013.482,-0.401,387.379,165.526,60.104,160.780
C08565=1013.476,-0.650,387.391,165.524,60.111,160.781
C08566=1013.472,-0.900,387.403,165.522,60.119,160.782
C08567=1013.468,-1.149,387.416,165.521,60.127,160.783
C08568=1013.462,-1.399,387.428,165.519,60.135,160.784
C08569=1013.458,-1.649,387.440,165.515,60.143,160.784
C08570=1013.453,-1.898,387.453,165.514,60.151,160.785
C08571=1013.449,-2.148,387.466,165.512,60.159,160.786
C08572=1013.444,-2.397,387.477,165.510,60.166,160.787
C08573=1013.439,-2.647,387.490,165.508,60.174,160.788
C08574=1013.435,-2.897,387.502,165.506,60.181,160.789
C08575=1013.430,-3.146,387.514,165.504,60.189,160.790
C08576=1013.425,-3.396,387.527,165.502,60.197,160.791
C08577=1013.421,-3.646,387.539,165.500,60.204,160.792
C08578=1013.416,-3.895,387.552,165.497,60.213,160.793
C08579=1013.411,-4.145,387.564,165.495,60.220,160.793
C08580=1013.407,-4.395,387.576,165.493,60.228,160.795
C08581=1013.403,-4.645,387.588,165.491,60.236,160.795
C08582=1013.397,-4.894,387.601,165.489,60.244,160.796
C08583=1013.393,-5.144,387.613,165.487,60.252,160.797
C08584=1013.388,-5.394,387.624,165.485,60.259,160.798
C08585=1013.382,-5.670,387.638,165.483,60.268,160.799
C08586=1013.377,-5.946,387.650,165.480,60.277,160.800
C08587=1013.372,-6.223,387.664,165.477,60.285,160.801
C08588=1013.367,-6.500,387.677,165.476,60.294,160.803
C08589=1013.362,-6.749,387.689,165.473,60.302,160.803
C08590=1013.357,-6.999,387.700,165.471,60.310,160.804
C08591=1013.352,-7.249,387.712,165.469,60.317,160.805
C08592=1013.347,-7.499,387.724,165.467,60.325,160.806
C08593=1013.343,-7.748,387.737,165.466,60.333,160.807
C08594=1013.338,-7.998,387.748,165.463,60.340,160.808
C08595=1013.333,-8.248,387.760,165.461,60.348,160.809
C08596=1013.329,-8.498,387.772,165.459,60.356,160.810
C08597=1013.324,-8.746,387.783,165.457,60.363,160.810
C08598=1013.319,-8.996,387.795,165.455,60.371,160.811
C08599=1013.315,-9.246,387.807,165.453,60.378,160.812
C08600=1013.310,-9.496,387.819,165.451,60.386,160.813
C08601=1013.304,-9.745,387.831,165.449,60.393,160.814
C08602=1013.300,-9.995,387.843,165.446,60.401,160.815
C08603=1013.295,-10.245,387.854,165.445,60.409,160.816
C08604=1013.290,-10.495,387.866,165.442,60.416,160.817
C08605=1013.286,-10.744,387.878,165.441,60.424,160.818
C08606=1013.281,-10.994,387.890,165.438,60.431,160.818
C08607=1013.276,-11.243,387.901,165.436,60.439,160.819
C08608=1013.272,-11.494,387.913,165.434,60.446,160.820
C08609=1013.267,-11.743,387.925,165.432,60.454,160.821
C08610=1013.262,-11.993,387.937,165.430,60.461,160.822
C08611=1013.257,-12.243,387.949,165.428,60.469,160.822
C08612=1013.253,-12.492,387.960,165.425,60.476,160.823
C08613=1013.248,-12.742,387.971,165.424,60.483,160.824
C08614=1013.244,-12.992,387.983,165.422,60.491,160.825
C08615=1013.239,-13.241,387.995,165.420,60.498,160.826
C08616=1013.233,-13.491,388.007,165.418,60.505,160.827
C08617=1013.229,-13.741,388.019,165.415,60.513,160.827
C08618=1013.225,-13.990,388.030,165.413,60.520,160.828
C08619=1013.220,-14.240,388.042,165.411,60.527,160.829
C08620=1013.215,-14.490,388.054,165.409,60.534,160.830
C08621=1013.210,-14.740,388.065,165.407,60.541,160.831
C08622=1013.205,-14.989,388.077,165.405,60.549,160.831
C08623=1013.201,-15.238,388.089,165.402,60.556,160.832
C08624=1013.196,-15.488,388.101,165.400,60.563,160.833
C08625=1013.191,-15.738,388.112,165.399,60.570,160.834
C08626=1013.187,-15.988,388.124,165.397,60.578,160.834
C08627=1013.182,-16.238,388.136,165.394,60.585,160.835
C08628=1013.178,-16.487,388.147,165.392,60.592,160.836
C08629=1013.173,-16.737,388.158,165.391,60.599,160.837
C08630=1013.168,-16.986,388.170,165.389,60.607,160.838
C08631=1013.163,-17.236,388.181,165.387,60.614,160.839
C08632=1013.159,-17.486,388.192,165.385,60.622,160.840
C08633=1013.154,-17.736,388.204,165.382,60.629,160.840
C08634=1013.149,-17.986,388.215,165.381,60.636,160.841
C08635=1013.144,-18.236,388.227,165.379,60.643,160.842
C08636=1013.140,-18.485,388.238,165.376,60.650,160.843
C08637=1013.135,-18.735,388.249,165.373,60.657,160.843
C08638=1013.130,-18.984,388.261,165.372,60.664,160.844
C08639=1013.125,-19.234,388.272,165.370,60.671,160.845
C08640=1013.121,-19.483,388.283,165.368,60.679,160.846
C08641=1013.116,-19.734,388.294,165.365,60.686,160.846
C08642=1013.111,-19.983,388.305,165.364,60.693,160.847
C08643=1013.106,-20.233,388.317,165.362,60.700,160.848
C08644=1013.101,-20.482,388.328,165.360,60.707,160.849
C08645=1013.096,-20.732,388.340,165.358,60.713,160.849
C08646=1013.092,-20.981,388.351,165.355,60.721,160.850
C08647=1013.087,-21.232,388.361,165.353,60.728,160.851
C08648=1013.082,-21.481,388.373,165.352,60.735,160.852
C08649=1013.079,-21.695,388.383,165.350,60.741,160.852
C08650=1013.074,-21.910,388.393,165.347,60.746,160.853
C08651=1013.070,-22.125,388.402,165.345,60.753,160.853
C08652=1013.066,-22.339,388.412,165.345,60.758,160.854
C08653=1013.063,-22.554,388.422,165.343,60.764,160.855
C08654=1013.058,-22.768,388.431,165.341,60.770,160.855
C08655=1013.054,-22.982,388.441,165.339,60.777,160.856
C08656=1013.051,-23.196,388.450,165.337,60.783,160.857
C08657=1013.046,-23.446,388.462,165.335,60.789,160.857
C08658=1013.041,-23.696,388.473,165.333,60.796,160.858
C08659=1013.037,-23.946,388.484,165.331,60.802,160.859
C08660=1013.032,-24.196,388.495,165.329,60.810,160.859
C08661=1013.027,-24.445,388.506,165.327,60.816,160.860
C08662=1013.022,-24.694,388.518,165.324,60.823,160.861
C08663=1013.017,-24.944,388.529,165.323,60.830,160.862
C08664=1013.013,-25.194,388.539,165.320,60.836,160.862
C08665=1013.008,-25.444,388.551,165.318,60.843,160.863
C08666=1013.004,-25.694,388.563,165.317,60.849,160.864
C08667=1013.000,-25.944,388.573,165.314,60.856,160.864
C08668=1012.995,-26.193,388.585,165.313,60.863,160.865
C08669=1012.990,-26.443,388.596,165.310,60.869,160.865
C08670=1012.985,-26.692,388.607,165.309,60.876,160.866
C08671=1012.981,-26.943,388.618,165.307,60.882,160.867
C08672=1012.976,-27.192,388.629,165.304,60.889,160.867
C08673=1012.971,-27.442,388.641,165.303,60.896,160.868
C08674=1012.966,-27.692,388.652,165.300,60.902,160.869
C08675=1012.962,-27.941,388.663,165.298,60.909,160.869
C08676=1012.957,-28.192,388.673,165.297,60.915,160.870
C08677=1012.953,-28.441,388.684,165.294,60.922,160.871
C08678=1012.948,-28.691,388.695,165.292,60.928,160.871
C08679=1012.943,-28.940,388.706,165.290,60.936,160.872
C08680=1012.938,-29.190,388.717,165.288,60.942,160.873
C08681=1012.933,-29.440,388.728,165.286,60.948,160.873
C08682=1012.929,-29.690,388.738,165.284,60.955,160.874
C08683=1012.924,-29.939,388.749,165.282,60.961,160.875
C08684=1012.920,-30.189,388.760,165.280,60.967,160.875
C08685=1012.915,-30.439,388.771,165.277,60.974,160.876
C08686=1012.910,-30.688,388.781,165.276,60.981,160.877
C08687=1012.905,-30.938,388.792,165.274,60.987,160.877
C08688=1012.901,-31.188,388.803,165.271,60.994,160.878
C08689=1012.896,-31.438,388.814,165.269,61.000,160.878
C08690=1012.891,-31.687,388.824,165.267,61.006,160.879
C08691=1012.886,-31.937,388.836,165.265,61.013,160.880
C08692=1012.882,-32.186,388.846,165.263,61.019,160.880
C08693=1012.877,-32.437,388.857,165.261,61.025,160.881
C08694=1012.873,-32.686,388.868,165.259,61.032,160.882
C08695=1012.867,-32.936,388.878,165.256,61.038,160.882
C08696=1012.863,-33.185,388.889,165.255,61.044,160.883
C08697=1012.858,-33.436,388.900,165.253,61.050,160.883
C08698=1012.854,-33.685,388.910,165.251,61.057,160.884
C08699=1012.848,-33.935,388.921,165.249,61.063,160.884
C08700=1012.844,-34.185,388.931,165.247,61.069,160.885
C08701=1012.841,-22.372,387.993,165.323,61.003,160.896
C08702=1012.845,-22.157,387.983,165.325,60.998,160.896
C08703=1012.850,-21.942,387.974,165.327,60.992,160.895
C08704=1012.853,-21.727,387.964,165.329,60.986,160.895
C08705=1012.857,-21.512,387.954,165.330,60.980,160.894
C08706=1012.861,-21.263,387.943,165.333,60.974,160.894
C08707=1012.866,-21.013,387.932,165.334,60.967,160.893
C08708=1012.871,-20.763,387.920,165.336,60.961,160.892
C08709=1012.876,-20.514,387.909,165.338,60.954,160.891
C08710=1012.881,-20.263,387.898,165.340,60.947,160.891
C08711=1012.886,-20.014,387.887,165.342,60.940,160.890
C08712=1012.890,-19.765,387.876,165.344,60.934,160.889
C08713=1012.895,-19.515,387.864,165.346,60.927,160.889
C08714=1012.900,-19.265,387.853,165.348,60.920,160.888
C08715=1012.904,-19.015,387.843,165.351,60.913,160.887
C08716=1012.909,-18.765,387.831,165.352,60.907,160.887
C08717=1012.914,-18.516,387.820,165.355,60.900,160.886
C08718=1012.919,-18.266,387.808,165.356,60.893,160.885
C08719=1012.923,-18.017,387.797,165.359,60.886,160.885
C08720=1012.928,-17.767,387.786,165.360,60.879,160.884
C08721=1012.932,-17.516,387.774,165.362,60.872,160.883
C08722=1012.937,-17.267,387.763,165.364,60.866,160.882
C08723=1012.942,-17.017,387.752,165.366,60.859,160.881
C08724=1012.947,-16.767,387.740,165.369,60.851,160.881
C08725=1012.951,-16.518,387.729,165.370,60.844,160.880
C08726=1012.956,-16.269,387.718,165.373,60.838,160.879
C08727=1012.961,-16.019,387.706,165.374,60.831,160.878
C08728=1012.965,-15.769,387.694,165.376,60.824,160.878
C08729=1012.970,-15.519,387.683,165.378,60.817,160.877
C08730=1012.975,-15.270,387.671,165.380,60.810,160.876
C08731=1012.979,-15.020,387.659,165.382,60.803,160.875
C08732=1012.984,-14.770,387.648,165.385,60.797,160.875
C08733=1012.989,-14.520,387.636,165.387,60.789,160.874
C08734=1012.993,-14.271,387.625,165.388,60.783,160.873
C08735=1012.998,-14.021,387.613,165.390,60.775,160.872
C08736=1013.003,-13.771,387.602,165.392,60.769,160.872
C08737=1013.007,-13.521,387.590,165.394,60.762,160.871
C08738=1013.012,-13.272,387.578,165.397,60.754,160.870
C08739=1013.017,-13.023,387.566,165.398,60.748,160.869
C08740=1013.021,-12.773,387.554,165.400,60.740,160.868
C08741=1013.026,-12.523,387.543,165.402,60.733,160.868
C08742=1013.031,-12.273,387.531,165.404,60.726,160.867
C08743=1013.035,-12.024,387.520,165.406,60.719,160.866
C08744=1013.040,-11.774,387.508,165.408,60.711,160.865
C08745=1013.045,-11.524,387.497,165.410,60.705,160.865
C08746=1013.049,-11.274,387.484,165.412,60.698,160.864
C08747=1013.054,-11.025,387.473,165.415,60.691,160.863
C08748=1013.059,-10.776,387.461,165.417,60.683,160.862
C08749=1013.063,-10.525,387.449,165.418,60.677,160.861
C08750=1013.068,-10.276,387.438,165.420,60.668,160.860
C08751=1013.073,-10.026,387.426,165.422,60.661,160.859
C08752=1013.078,-9.776,387.414,165.424,60.654,160.859
C08753=1013.083,-9.527,387.402,165.427,60.646,160.858
C08754=1013.087,-9.277,387.391,165.428,60.640,160.857
C08755=1013.091,-9.027,387.379,165.430,60.632,160.856
C08756=1013.096,-8.778,387.367,165.432,60.625,160.855
C08757=1013.101,-8.528,387.355,165.435,60.618,160.855
C08758=1013.106,-8.278,387.343,165.436,60.610,160.854
C08759=1013.111,-8.028,387.332,165.439,60.602,160.853
C08760=1013.115,-7.778,387.320,165.441,60.595,160.852
C08761=1013.119,-7.529,387.309,165.442,60.588,160.851
C08762=1013.125,-7.280,387.296,165.444,60.580,160.850
C08763=1013.129,-7.030,387.284,165.446,60.573,160.849
C08764=1013.134,-6.780,387.273,165.448,60.566,160.849
C08765=1013.139,-6.530,387.261,165.451,60.558,160.848
C08766=1013.145,-6.254,387.248,165.453,60.550,160.847
C08767=1013.149,-5.977,387.235,165.455,60.542,160.846
C08768=1013.154,-5.701,387.222,165.458,60.533,160.845
C08769=1013.160,-5.425,387.208,165.460,60.524,160.844
C08770=1013.165,-5.175,387.197,165.462,60.517,160.843
C08771=1013.169,-4.925,387.185,165.464,60.509,160.842
C08772=1013.174,-4.675,387.173,165.466,60.501,160.841
C08773=1013.179,-4.426,387.160,165.467,60.494,160.840
C08774=1013.183,-4.177,387.149,165.469,60.487,160.839
C08775=1013.188,-3.927,387.136,165.471,60.479,160.838
C08776=1013.192,-3.677,387.124,165.473,60.472,160.838
C08777=1013.197,-3.428,387.112,165.476,60.464,160.837
C08778=1013.202,-3.178,387.100,165.477,60.456,160.836
C08779=1013.206,-2.928,387.087,165.480,60.449,160.835
C08780=1013.211,-2.678,387.075,165.482,60.442,160.834
C08781=1013.216,-2.429,387.063,165.484,60.434,160.833
C08782=1013.221,-2.179,387.050,165.486,60.426,160.832
C08783=1013.225,-1.929,387.038,165.488,60.418,160.831
C08784=1013.229,-1.680,387.025,165.490,60.411,160.831
C08785=1013.234,-1.430,387.014,165.492,60.404,160.830
C08786=1013.239,-1.181,387.001,165.494,60.396,160.829
C08787=1013.243,-0.930,386.989,165.496,60.389,160.828
C08788=1013.248,-0.681,386.976,165.498,60.380,160.827
C08789=1013.253,-0.432,386.964,165.500,60.373,160.826
C08790=1013.257,-0.182,386.952,165.502,60.365,160.825
C08791=1013.262,0.068,386.939,165.504,60.358,160.824
C08792=1013.267,0.318,386.928,165.506,60.350,160.823
C08793=1013.271,0.567,386.915,165.508,60.342,160.822
C08794=1013.276,0.817,386.902,165.510,60.335,160.821
C08795=1013.280,1.067,386.890,165.512,60.327,160.820
C08796=1013.286,1.316,386.878,165.514,60.319,160.819
C08797=1013.290,1.566,386.866,165.516,60.311,160.818
C08798=1013.294,1.816,386.853,165.517,60.303,160.817
C08799=1013.299,2.065,386.840,165.521,60.295,160.817
C08800=1013.304,2.315,386.829,165.522,60.287,160.816
C08801=1013.309,2.564,386.816,165.524,60.279,160.815
C08802=1013.313,2.814,386.803,165.526,60.271,160.813
C08803=1013.318,3.064,386.792,165.528,60.264,160.813
C08804=1013.323,3.313,386.779,165.530,60.256,160.812
C08805=1013.327,3.563,386.766,165.532,60.248,160.811
C08806=1013.332,3.813,386.754,165.534,60.240,160.810
C08807=1013.337,4.062,386.742,165.536,60.232,160.809
C08808=1013.341,4.311,386.729,165.538,60.224,160.808
C08809=1013.346,4.562,386.717,165.540,60.216,160.807
C08810=1013.350,4.811,386.704,165.543,60.208,160.806
C08811=1013.356,5.061,386.692,165.544,60.200,160.805
C08812=1013.360,5.311,386.680,165.546,60.192,160.804
C08813=1013.365,5.561,386.667,165.548,60.184,160.803
C08814=1013.370,5.810,386.655,165.550,60.175,160.802
C08815=1013.375,6.059,386.642,165.552,60.167,160.801
C08816=1013.379,6.309,386.630,165.554,60.159,160.800
C08817=1013.384,6.559,386.617,165.556,60.151,160.799
C08818=1013.389,6.808,386.605,165.558,60.143,160.798
C08819=1013.393,7.058,386.593,165.560,60.135,160.797
C08820=1013.398,7.308,386.580,165.563,60.126,160.796
C08821=1013.402,7.557,386.567,165.564,60.118,160.795
C08822=1013.408,7.807,386.555,165.566,60.110,160.794
C08823=1013.413,8.057,386.543,165.569,60.102,160.793
C08824=1013.417,8.307,386.530,165.570,60.094,160.792
C08825=1013.422,8.556,386.517,165.572,60.086,160.791
C08826=1013.427,8.805,386.505,165.575,60.077,160.790
C08827=1013.432,9.055,386.492,165.577,60.069,160.789
C08828=1013.436,9.305,386.480,165.579,60.061,160.788
C08829=1013.440,9.554,386.467,165.581,60.053,160.787
C08830=1013.446,9.833,386.453,165.583,60.043,160.785
C08831=1013.452,10.112,386.439,165.585,60.034,160.784
C08832=1013.457,10.390,386.425,165.588,60.024,160.783
C08833=1013.463,10.669,386.411,165.590,60.015,160.782
C08834=1013.467,10.919,386.399,165.592,60.007,160.781
C08835=1013.472,11.168,386.387,165.595,59.998,160.780
C08836=1013.477,11.417,386.374,165.596,59.990,160.778
C08837=1013.482,11.668,386.361,165.598,59.981,160.777
C08838=1013.486,11.917,386.348,165.600,59.973,160.776
C08839=1013.491,12.167,386.337,165.603,59.965,160.776
C08840=1013.496,12.416,386.324,165.604,59.956,160.774
C08841=1013.501,12.666,386.311,165.607,59.948,160.773
C08842=1013.506,12.916,386.298,165.609,59.938,160.772
C08843=1013.510,13.166,386.285,165.611,59.930,160.771
C08844=1013.515,13.415,386.272,165.612,59.923,160.770
C08845=1013.519,13.664,386.260,165.615,59.914,160.769
C08846=1013.525,13.915,386.246,165.616,59.905,160.768
C08847=1013.529,14.164,386.234,165.619,59.897,160.767
C08848=1013.534,14.414,386.221,165.621,59.889,160.766
C08849=1013.538,14.663,386.208,165.624,59.880,160.765
C08850=1013.543,14.913,386.195,165.625,59.872,160.763
C08851=1013.548,15.163,386.182,165.627,59.863,160.763
C08852=1013.553,15.412,386.169,165.629,59.855,160.761
C08853=1013.557,15.662,386.157,165.631,59.846,160.760
C08854=1013.562,15.911,386.143,165.633,59.838,160.759
C08855=1013.567,16.161,386.130,165.635,59.829,160.758
C08856=1013.572,16.410,386.117,165.637,59.821,160.757
C08857=1013.576,16.660,386.104,165.639,59.812,160.756
C08858=1013.581,16.909,386.092,165.642,59.803,160.755
C08859=1013.586,17.160,386.078,165.644,59.795,160.754
C08860=1013.591,17.409,386.066,165.646,59.786,160.753
C08861=1013.595,17.659,386.053,165.648,59.778,160.752
C08862=1013.600,17.908,386.040,165.650,59.769,160.750
C08863=1013.605,18.158,386.026,165.652,59.761,160.749
C08864=1013.610,18.407,386.013,165.654,59.752,160.748
C08865=1013.614,18.657,386.001,165.656,59.743,160.747
C08866=1013.619,18.907,385.987,165.658,59.735,160.746
C08867=1013.623,19.157,385.974,165.660,59.726,160.745
C08868=1013.628,19.406,385.961,165.662,59.718,160.744
C08869=1013.634,19.656,385.947,165.664,59.709,160.743
C08870=1013.638,19.905,385.935,165.667,59.700,160.742
C08871=1013.642,20.155,385.921,165.668,59.692,160.740
C08872=1013.647,20.405,385.908,165.671,59.683,160.739
C08873=1013.652,20.654,385.895,165.673,59.674,160.738
C08874=1013.657,20.904,385.882,165.675,59.666,160.737
C08875=1013.662,21.154,385.869,165.677,59.657,160.736
C08876=1013.666,21.404,385.855,165.678,59.648,160.735
C08877=1013.670,21.652,385.842,165.681,59.640,160.734
C08878=1013.675,21.902,385.829,165.683,59.631,160.733
C08879=1013.680,22.152,385.816,165.685,59.621,160.731
C08880=1013.685,22.401,385.802,165.687,59.614,160.730
C08881=1013.690,22.650,385.790,165.689,59.604,160.729
C08882=1013.694,22.901,385.776,165.692,59.595,160.728
C08883=1013.699,23.150,385.762,165.693,59.587,160.727
C08884=1013.704,23.400,385.749,165.696,59.578,160.726
C08885=1013.709,23.650,385.736,165.698,59.569,160.725
C08886=1013.714,23.898,385.723,165.700,59.560,160.723
C08887=1013.718,24.149,385.709,165.701,59.551,160.722
C08888=1013.723,24.398,385.696,165.704,59.543,160.721
C08889=1013.727,24.647,385.683,165.706,59.534,160.720
C08890=1013.733,24.897,385.670,165.708,59.524,160.719
C08891=1013.737,25.147,385.657,165.710,59.516,160.717
C08892=1013.742,25.397,385.643,165.712,59.507,160.716
C08893=1013.746,25.646,385.630,165.714,59.498,160.715
C08894=1013.752,25.926,385.615,165.717,59.488,160.714
C08895=1013.757,26.207,385.600,165.719,59.478,160.713
C08896=1013.763,26.486,385.585,165.722,59.468,160.711
C08897=1013.768,26.766,385.569,165.723,59.458,160.710
C08898=1013.773,27.017,385.556,165.725,59.449,160.709
C08899=1013.777,27.266,385.543,165.728,59.440,160.707
C08900=1013.781,27.515,385.529,165.730,59.431,160.706
C08901=1013.787,27.765,385.516,165.733,59.422,160.705
C08902=1013.791,28.015,385.502,165.734,59.413,160.704
C08903=1013.796,28.264,385.488,165.736,59.404,160.703
C08904=1013.800,28.514,385.475,165.739,59.395,160.702
C08905=1013.806,28.764,385.461,165.741,59.386,160.701
C08906=1013.810,29.013,385.448,165.742,59.377,160.699
C08907=1013.815,29.263,385.434,165.744,59.368,160.698
C08908=1013.819,29.512,385.421,165.747,59.359,160.697
C08909=1013.824,29.762,385.407,165.749,59.350,160.696
C08910=1013.829,30.011,385.393,165.751,59.341,160.695
C08911=1013.833,30.261,385.380,165.753,59.332,160.693
C08912=1013.838,30.511,385.366,165.755,59.323,160.692
C08913=1013.842,30.760,385.352,165.757,59.314,160.691
C08914=1013.848,31.010,385.338,165.759,59.305,160.690
C08915=1013.852,31.259,385.325,165.761,59.296,160.688
C08916=1013.857,31.509,385.311,165.764,59.287,160.687
C08917=1013.862,31.758,385.298,165.766,59.278,160.686
C08918=1013.867,32.008,385.283,165.768,59.269,160.685
C08919=1013.871,32.258,385.270,165.770,59.259,160.684
C08920=1013.876,32.507,385.256,165.772,59.251,160.682
C08921=1013.881,32.756,385.242,165.774,59.242,160.681
C08922=1013.885,33.007,385.229,165.776,59.233,160.680
C08923=1013.890,33.256,385.215,165.779,59.224,160.679
C08924=1013.895,33.505,385.201,165.780,59.214,160.677
C08925=1013.899,33.755,385.188,165.783,59.205,160.676
C08926=1013.905,34.005,385.174,165.785,59.196,160.675
C08927=1013.909,34.254,385.160,165.787,59.186,160.674
C08928=1013.914,34.504,385.147,165.789,59.177,160.673
C08929=1013.918,34.753,385.133,165.791,59.168,160.671
C08930=1013.924,35.003,385.119,165.793,59.158,160.670
C08931=1013.928,35.253,385.106,165.796,59.149,160.669
C08932=1013.933,35.502,385.092,165.798,59.140,160.668
C08933=1013.937,35.751,385.078,165.800,59.130,160.666
C08934=1013.942,36.002,385.064,165.802,59.121,160.665
C08935=1013.946,36.251,385.050,165.804,59.112,160.664
C08936=1013.952,36.500,385.036,165.807,59.103,160.663
C08937=1013.957,36.750,385.022,165.808,59.093,160.662
C08938=1013.961,36.999,385.008,165.811,59.084,160.660
C08939=1013.966,37.249,384.994,165.813,59.075,160.659
C08940=1013.970,37.499,384.981,165.815,59.066,160.658
C08941=1013.975,37.749,384.966,165.818,59.057,160.657
C08942=1013.980,37.998,384.953,165.819,59.047,160.655
C08943=1013.984,38.247,384.938,165.822,59.038,160.654
C08944=1013.989,38.497,384.924,165.824,59.029,160.653
C08945=1013.993,38.747,384.910,165.826,59.019,160.652
C08946=1013.999,38.996,384.896,165.828,59.010,160.651
C08947=1014.003,39.245,384.882,165.830,59.001,160.649
C08948=1014.008,39.495,384.867,165.833,58.992,160.648
C08949=1014.013,39.745,384.853,165.834,58.982,160.647
C08950=1014.017,39.994,384.839,165.837,58.973,160.646
C08951=1014.022,40.244,384.825,165.839,58.964,160.644
C08952=1014.026,40.494,384.812,165.841,58.954,160.643
C08953=1014.031,40.743,384.798,165.843,58.945,160.642
C08954=1014.036,40.993,384.783,165.845,58.936,160.640
C08955=1014.040,41.242,384.769,165.847,58.926,160.639
C08956=1014.046,41.492,384.755,165.850,58.917,160.638
C08957=1014.050,41.741,384.741,165.851,58.908,160.637
C08958=1014.055,42.022,384.725,165.854,58.897,160.635
C08959=1014.061,42.301,384.709,165.856,58.886,160.634
C08960=1014.066,42.582,384.692,165.859,58.876,160.633
C08961=1014.071,42.863,384.676,165.862,58.866,160.631
C08962=1014.075,43.112,384.662,165.863,58.857,160.630
C08963=1014.080,43.362,384.648,165.865,58.848,160.628
C08964=1014.085,43.611,384.633,165.867,58.838,160.627
C08965=1014.089,43.860,384.619,165.869,58.829,160.626
C08966=1014.094,44.110,384.604,165.872,58.820,160.625
C08967=1014.099,44.360,384.590,165.875,58.810,160.624
C08968=1014.103,44.609,384.576,165.877,58.800,160.622
C08969=1014.108,44.859,384.560,165.879,58.791,160.621
C08970=1014.113,45.108,384.546,165.881,58.782,160.620
C08971=1014.117,45.358,384.532,165.883,58.773,160.619
C08972=1014.121,45.608,384.517,165.885,58.763,160.617
C08973=1014.126,45.857,384.503,165.887,58.754,160.616
C08974=1014.131,46.106,384.488,165.890,58.745,160.615
C08975=1014.135,46.356,384.474,165.892,58.735,160.613
C08976=1014.140,46.606,384.459,165.894,58.726,160.612
C08977=1014.144,46.855,384.445,165.896,58.716,160.611
C08978=1014.149,47.104,384.430,165.898,58.707,160.610
C08979=1014.154,47.354,384.415,165.900,58.697,160.608
C08980=1014.158,47.603,384.401,165.902,58.688,160.607
C08981=1014.163,47.853,384.387,165.905,58.678,160.606
C08982=1014.168,48.102,384.372,165.907,58.668,160.604
C08983=1014.173,48.352,384.357,165.910,58.659,160.603
C08984=1014.177,48.601,384.343,165.911,58.650,160.602
C08985=1014.182,48.851,384.329,165.914,58.641,160.601
C08986=1014.187,49.101,384.314,165.916,58.631,160.599
C08987=1014.191,49.351,384.299,165.917,58.621,160.598
C08988=1014.196,49.600,384.285,165.921,58.612,160.597
C08989=1014.200,49.850,384.270,165.923,58.602,160.596
C08990=1014.205,50.099,384.255,165.924,58.592,160.594
C08991=1014.210,50.349,384.241,165.927,58.583,160.593
C08992=1014.214,50.598,384.227,165.929,58.573,160.592
C08993=1014.219,50.847,384.212,165.931,58.564,160.590
C08994=1014.224,51.097,384.197,165.934,58.554,160.589
C08995=1014.228,51.347,384.182,165.936,58.544,160.588
C08996=1014.232,51.596,384.167,165.938,58.535,160.586
C08997=1014.237,51.846,384.153,165.940,58.525,160.585
C08998=1014.242,52.096,384.138,165.943,58.515,160.584
C08999=1014.247,52.345,384.123,165.945,58.506,160.583
C09000=1014.251,52.594,384.109,165.947,58.496,160.581
C09001=1014.256,52.844,384.095,165.949,58.486,160.580
C09002=1014.261,53.093,384.079,165.952,58.477,160.579
C09003=1014.266,53.343,384.065,165.954,58.467,160.577
C09004=1014.270,53.593,384.051,165.956,58.457,160.576
C09005=1014.275,53.842,384.036,165.958,58.448,160.574
C09006=1014.279,54.091,384.021,165.961,58.437,160.573
C09007=1014.285,54.341,384.006,165.962,58.428,160.572
C09008=1014.289,54.591,383.992,165.964,58.418,160.570
C09009=1014.294,54.841,383.977,165.968,58.409,160.569
C09010=1014.299,55.090,383.962,165.970,58.399,160.568
C09011=1014.303,55.339,383.948,165.971,58.389,160.567
C09012=1014.308,55.588,383.933,165.974,58.379,160.565
C09013=1014.313,55.838,383.918,165.976,58.369,160.564
C09014=1014.318,56.088,383.904,165.978,58.359,160.562
C09015=1014.323,56.337,383.889,165.981,58.349,160.561
C09016=1014.327,56.587,383.874,165.983,58.340,160.560
C09017=1014.332,56.836,383.859,165.985,58.330,160.558
C09018=1014.337,57.086,383.845,165.988,58.320,160.557
C09019=1014.342,57.335,383.830,165.990,58.310,160.556
C09020=1014.346,57.585,383.815,165.993,58.300,160.555
C09021=1014.351,57.835,383.801,165.995,58.290,160.553
C09022=1014.357,58.115,383.784,165.997,58.279,160.552
C09023=1014.362,58.394,383.767,166.000,58.268,160.550
C09024=1014.367,58.675,383.751,166.003,58.257,160.549
C09025=1014.372,58.956,383.734,166.004,58.245,160.547
C09026=1014.377,59.205,383.720,166.007,58.235,160.546
C09027=1014.382,59.455,383.704,166.009,58.226,160.544
C09028=1014.387,59.705,383.690,166.011,58.216,160.543
C09029=1014.392,59.954,383.675,166.014,58.206,160.542
C09030=1014.397,60.204,383.660,166.016,58.196,160.540
C09031=1014.401,60.452,383.645,166.019,58.186,160.539
C09032=1014.406,60.702,383.631,166.020,58.176,160.537
C09033=1014.411,60.951,383.616,166.023,58.165,160.536
C09034=1014.416,61.201,383.601,166.025,58.156,160.535
C09035=1014.421,61.451,383.586,166.028,58.146,160.533
C09036=1014.426,61.700,383.571,166.030,58.136,160.532
C09037=1014.430,61.950,383.557,166.033,58.126,160.531
C09038=1014.436,62.199,383.541,166.034,58.115,160.529
C09039=1014.440,62.449,383.527,166.037,58.105,160.528
C09040=1014.445,62.698,383.512,166.039,58.096,160.526
C09041=1014.449,62.948,383.497,166.042,58.085,160.525
C09042=1014.454,63.198,383.482,166.044,58.076,160.524
C09043=1014.459,63.447,383.466,166.046,58.066,160.522
C09044=1014.464,63.696,383.451,166.049,58.056,160.521
C09045=1014.468,63.946,383.436,166.051,58.046,160.520
C09046=1014.473,64.196,383.421,166.054,58.036,160.519
C09047=1014.478,64.445,383.405,166.056,58.026,160.517
C09048=1014.482,64.694,383.390,166.058,58.016,160.516
C09049=1014.487,64.944,383.376,166.061,58.006,160.514
C09050=1014.491,65.193,383.360,166.062,57.996,160.513
C09051=1014.496,65.442,383.345,166.066,57.986,160.512
C09052=1014.501,65.692,383.330,166.067,57.977,160.510
C09053=1014.506,65.941,383.314,166.069,57.967,160.509
C09054=1014.510,66.191,383.300,166.072,57.956,160.507
C09055=1014.515,66.441,383.284,166.074,57.946,160.506
C09056=1014.520,66.690,383.269,166.077,57.936,160.505
C09057=1014.525,66.939,383.253,166.079,57.927,160.503
C09058=1014.529,67.189,383.238,166.082,57.917,160.502
C09059=1014.534,67.438,383.222,166.084,57.907,160.501
C09060=1014.538,67.688,383.207,166.086,57.896,160.499
C09061=1014.543,67.938,383.192,166.088,57.886,160.498
C09062=1014.548,68.187,383.177,166.090,57.877,160.497
C09063=1014.553,68.436,383.161,166.093,57.867,160.495
C09064=1014.557,68.686,383.146,166.095,57.857,160.494
C09065=1014.562,68.935,383.130,166.098,57.846,160.492
C09066=1014.566,69.185,383.115,166.100,57.837,160.491
C09067=1014.571,69.434,383.099,166.103,57.827,160.490
C09068=1014.576,69.684,383.084,166.105,57.817,160.488
C09069=1014.581,69.934,383.068,166.108,57.807,160.487
C09070=1014.585,70.183,383.052,166.109,57.796,160.486
C09071=1014.591,70.433,383.037,166.111,57.787,160.484
C09072=1014.595,70.682,383.021,166.115,57.777,160.483
C09073=1014.599,70.932,383.006,166.117,57.767,160.482
C09074=1014.604,71.181,382.990,166.119,57.756,160.480
C09075=1014.608,71.431,382.975,166.121,57.747,160.479
C09076=1014.614,71.680,382.960,166.124,57.737,160.478
C09077=1014.618,71.929,382.944,166.126,57.727,160.476
C09078=1014.623,72.179,382.929,166.129,57.716,160.475
C09079=1014.627,72.428,382.913,166.131,57.707,160.473
C09080=1014.631,72.678,382.897,166.134,57.697,160.472
C09081=1014.637,72.927,382.882,166.136,57.687,160.471
C09082=1014.641,73.177,382.866,166.138,57.676,160.469
C09083=1014.646,73.426,382.851,166.140,57.666,160.468
C09084=1014.650,73.675,382.834,166.144,57.656,160.467
C09085=1014.655,73.925,382.818,166.145,57.646,160.465
C09086=1014.661,74.206,382.801,166.149,57.635,160.464
C09087=1014.666,74.486,382.784,166.150,57.623,160.462
C09088=1014.671,74.766,382.766,166.154,57.612,160.461
C09089=1014.676,75.046,382.748,166.156,57.601,160.459
C09090=1014.681,75.295,382.733,166.159,57.591,160.458
C09091=1014.686,75.545,382.718,166.161,57.580,160.456
C09092=1014.691,75.795,382.701,166.164,57.570,160.455
C09093=1014.696,76.045,382.686,166.167,57.560,160.454
C09094=1014.700,76.294,382.670,166.168,57.550,160.452
C09095=1014.705,76.543,382.654,166.171,57.540,160.451
C09096=1014.709,76.793,382.638,166.173,57.530,160.449
C09097=1014.714,77.042,382.623,166.176,57.519,160.448
C09098=1014.718,77.292,382.607,166.178,57.510,160.447
C09099=1014.723,77.541,382.590,166.181,57.499,160.445
C09100=1014.728,77.791,382.575,166.183,57.490,160.444
C09101=1014.732,78.040,382.559,166.186,57.480,160.443
C09102=1014.737,78.289,382.542,166.187,57.469,160.441
C09103=1014.741,78.539,382.527,166.191,57.459,160.440
C09104=1014.746,78.788,382.511,166.193,57.450,160.438
C09105=1014.751,79.038,382.495,166.195,57.439,160.437
C09106=1014.755,79.287,382.479,166.197,57.429,160.435
C09107=1014.760,79.537,382.463,166.201,57.419,160.434
C09108=1014.764,79.786,382.447,166.202,57.409,160.433
C09109=1014.769,80.035,382.431,166.205,57.399,160.431
C09110=1014.773,80.285,382.415,166.207,57.389,160.430
C09111=1014.778,80.535,382.398,166.210,57.379,160.429
C09112=1014.783,80.784,382.383,166.212,57.369,160.427
C09113=1014.788,81.033,382.367,166.215,57.358,160.426
C09114=1014.792,81.283,382.351,166.217,57.349,160.424
C09115=1014.796,81.532,382.335,166.219,57.338,160.423
C09116=1014.802,81.782,382.318,166.223,57.328,160.422
C09117=1014.806,82.031,382.302,166.224,57.318,160.420
C09118=1014.811,82.280,382.286,166.227,57.308,160.419
C09119=1014.815,82.530,382.270,166.229,57.297,160.417
C09120=1014.819,82.779,382.254,166.232,57.287,160.416
C09121=1014.825,83.029,382.238,166.235,57.277,160.415
C09122=1014.829,83.278,382.222,166.237,57.267,160.413
C09123=1014.834,83.527,382.206,166.240,57.256,160.412
C09124=1014.838,83.777,382.190,166.242,57.247,160.411
C09125=1014.844,84.027,382.173,166.244,57.236,160.409
C09126=1014.848,84.276,382.157,166.248,57.226,160.408
C09127=1014.852,84.526,382.142,166.249,57.216,160.406
